LIN {X 0,Y 311.032,Z 352.826,A -85,B 0,C 180,E1 -15949.126,E2 -15949.126} C_VEL
LIN {X 0,Y 312.836,Z 341.868,A -85,B 0,C 180,E1 -15950.55,E2 -15950.55} C_VEL
LIN {X 0,Y 314.374,Z 331.182,A -85,B 0,C 180,E1 -15951.646,E2 -15951.646} C_VEL
LIN {X 0,Y 315.929,Z 318.395,A -85,B 0,C 180,E1 -15952.652,E2 -15952.652} C_VEL
LIN {X 0,Y 317.171,Z 305.489,A -85,B 0,C 180,E1 -15953.377,E2 -15953.377} C_VEL
LIN {X 0,Y 317.99,Z 291.946,A -85,B 0,C 180,E1 -15953.864,E2 -15953.864} C_VEL
LIN {X 0,Y 319.812,Z 229.515,A -85,B 0,C 180,E1 -15955.377,E2 -15955.377} C_VEL
LIN {X 0,Y 316.738,Z 210.082,A -85,B 0,C 180,E1 -15956.219,E2 -15956.219} C_VEL
LIN {X 0,Y 313.412,Z 194.203,A -85,B 0,C 180,E1 -15957.021,E2 -15957.021} C_VEL
LIN {X 0,Y 310.374,Z 186.88,A -85,B 0,C 180,E1 -15957.598,E2 -15957.598} C_VEL
LIN {X 0,Y 308.319,Z 176.835,A -85,B 0,C 180,E1 -15960.855,E2 -15960.855} C_VEL
LIN {X 0,Y 305.949,Z 167.212,A -85,B 0,C 180,E1 -15964.212,E2 -15964.212} C_VEL
LIN {X 0,Y 305.464,Z 165.436,A -85,B 0,C 180,E1 -15964.901,E2 -15964.901} C_VEL
LIN {X 0,Y 305.434,Z 165.44,A -85,B 0,C 180,E1 -15968.525,E2 -15968.525} C_VEL
LIN {X 0,Y 305.435,Z 165.44,A -85,B 0,C 180,E1 -15972.582,E2 -15972.582} C_VEL
LIN {X 0,Y 305.422,Z 165.442,A -85,B 0,C 180,E1 -15976.344,E2 -15976.344} C_VEL
LIN {X 0,Y 305.411,Z 165.436,A -85,B 0,C 180,E1 -15979.885,E2 -15979.885} C_VEL
LIN {X 0,Y 305.464,Z 165.428,A -85,B 0,C 180,E1 -15983.637,E2 -15983.637} C_VEL
LIN {X 0,Y 305.467,Z 165.428,A -85,B 0,C 180,E1 -15986.483,E2 -15986.483} C_VEL
LIN {X 0,Y 305.419,Z 165.437,A -85,B 0,C 180,E1 -15989.586,E2 -15989.586} C_VEL
LIN {X 0,Y 305.442,Z 165.436,A -85,B 0,C 180,E1 -15992.601,E2 -15992.601} C_VEL
LIN {X 0,Y 305.441,Z 165.427,A -85,B 0,C 180,E1 -15995.533,E2 -15995.533} C_VEL
LIN {X 0,Y 305.475,Z 165.42,A -85,B 0,C 180,E1 -15999.812,E2 -15999.812} C_VEL
LIN {X 0,Y 305.494,Z 165.421,A -85,B 0,C 180,E1 -16003.975,E2 -16003.975} C_VEL
LIN {X 0,Y 305.557,Z 165.423,A -85,B 0,C 180,E1 -16006.703,E2 -16006.703} C_VEL
LIN {X 0,Y 305.766,Z 165.394,A -85,B 0,C 180,E1 -16011.249,E2 -16011.249} C_VEL
LIN {X 0,Y 305.798,Z 165.379,A -85,B 0,C 180,E1 -16013.401,E2 -16013.401} C_VEL
LIN {X 0,Y 305.937,Z 165.369,A -85,B 0,C 180,E1 -16018.684,E2 -16018.684} C_VEL
LIN {X 0,Y 305.937,Z 165.369,A -85,B 0,C 180,E1 -16021.316,E2 -16021.316} C_VEL
LIN {X 0,Y 305.788,Z 165.391,A -85,B 0,C 180,E1 -16026.599,E2 -16026.599} C_VEL
LIN {X 0,Y 305.697,Z 165.4,A -85,B 0,C 180,E1 -16029.261,E2 -16029.261} C_VEL
LIN {X 0,Y 305.573,Z 165.418,A -85,B 0,C 180,E1 -16033.297,E2 -16033.297} C_VEL
LIN {X 0,Y 305.514,Z 165.427,A -85,B 0,C 180,E1 -16036.025,E2 -16036.025} C_VEL
LIN {X 0,Y 305.475,Z 165.431,A -85,B 0,C 180,E1 -16040.188,E2 -16040.188} C_VEL
LIN {X 0,Y 305.443,Z 165.439,A -85,B 0,C 180,E1 -16044.467,E2 -16044.467} C_VEL
LIN {X 0,Y 305.454,Z 165.451,A -85,B 0,C 180,E1 -16047.213,E2 -16047.213} C_VEL
LIN {X 0,Y 307.467,Z 173.471,A -85,B 0,C 180,E1 -16050.15,E2 -16050.15} C_VEL
LIN {X 0,Y 315.579,Z 190.715,A -85,B 0,C 180,E1 -16051.565,E2 -16051.565} C_VEL
LIN {X 0,Y 319.554,Z 201.138,A -85,B 0,C 180,E1 -16052.271,E2 -16052.271} C_VEL
LIN {X 0,Y 320.576,Z 206.188,A -85,B 0,C 180,E1 -16052.511,E2 -16052.511} C_VEL
LIN {X 0,Y 318.103,Z 281.171,A -85,B 0,C 180,E1 -16054.335,E2 -16054.335} C_VEL
LIN {X 0,Y 317.204,Z 294.383,A -85,B 0,C 180,E1 -16054.902,E2 -16054.902} C_VEL
LIN {X 0,Y 316.114,Z 307.547,A -85,B 0,C 180,E1 -16055.758,E2 -16055.758} C_VEL
LIN {X 0,Y 314.765,Z 318.834,A -85,B 0,C 180,E1 -16056.743,E2 -16056.743} C_VEL
LIN {X 0,Y 313.128,Z 330.027,A -85,B 0,C 180,E1 -16057.991,E2 -16057.991} C_VEL
LIN {X 0,Y 311.462,Z 340.557,A -85,B 0,C 180,E1 -16059.476,E2 -16059.476} C_VEL
LIN {X 0,Y 309.82,Z 349.922,A -85,B 0,C 180,E1 -16061.136,E2 -16061.136} C_VEL
LIN {X 0,Y 308.123,Z 358.925,A -85,B 0,C 180,E1 -16063.122,E2 -16063.122} C_VEL
LIN {X 0,Y 306.651,Z 366.582,A -85,B 0,C 180,E1 -16065.274,E2 -16065.274} C_VEL
LIN {X 0,Y 305.538,Z 372.451,A -85,B 0,C 180,E1 -16067.398,E2 -16067.398} C_VEL
LIN {X 0,Y 304.642,Z 377.4,A -85,B 0,C 180,E1 -16069.762,E2 -16069.762} C_VEL
LIN {X 0,Y 304.056,Z 380.454,A -85,B 0,C 180,E1 -16071.803,E2 -16071.803} C_VEL
LIN {X 0,Y 303.595,Z 382.701,A -85,B 0,C 180,E1 -16074.118,E2 -16074.118} C_VEL
LIN {X 0,Y 303.326,Z 383.694,A -85,B 0,C 180,E1 -16076.524,E2 -16076.524} C_VEL
LIN {X 0,Y 303.317,Z 383.355,A -85,B 0,C 180,E1 -16079.016,E2 -16079.016} C_VEL
LIN {X 0,Y 303.5,Z 381.483,A -85,B 0,C 180,E1 -16081.637,E2 -16081.637} C_VEL
LIN {X 0,Y 303.941,Z 378.457,A -85,B 0,C 180,E1 -16083.938,E2 -16083.938} C_VEL
LIN {X 0,Y 304.435,Z 374.226,A -85,B 0,C 180,E1 -16086.172,E2 -16086.172} C_VEL
LIN {X 0,Y 305.054,Z 368.671,A -85,B 0,C 180,E1 -16088.369,E2 -16088.369} C_VEL
LIN {X 0,Y 305.932,Z 362.172,A -85,B 0,C 180,E1 -16090.369,E2 -16090.369} C_VEL
LIN {X 0,Y 307.109,Z 354.061,A -85,B 0,C 180,E1 -16092.349,E2 -16092.349} C_VEL
LIN {X 0,Y 308.333,Z 345.04,A -85,B 0,C 180,E1 -16094.126,E2 -16094.126} C_VEL
LIN {X 0,Y 309.623,Z 335.151,A -85,B 0,C 180,E1 -16095.694,E2 -16095.694} C_VEL
LIN {X 0,Y 310.97,Z 323.96,A -85,B 0,C 180,E1 -16097.104,E2 -16097.104} C_VEL
LIN {X 0,Y 312.192,Z 311.78,A -85,B 0,C 180,E1 -16098.31,E2 -16098.31} C_VEL
LIN {X 0,Y 313.171,Z 299.062,A -85,B 0,C 180,E1 -16099.249,E2 -16099.249} C_VEL
LIN {X 0,Y 314.061,Z 285.587,A -85,B 0,C 180,E1 -16099.942,E2 -16099.942} C_VEL
LIN {X 0,Y 314.631,Z 272.038,A -85,B 0,C 180,E1 -16100.359,E2 -16100.359} C_VEL
LIN {X 0,Y 316.256,Z 204.158,A -85,B 0,C 180,E1 -16101.974,E2 -16101.974} C_VEL
LIN {X 0,Y 313.704,Z 190.916,A -85,B 0,C 180,E1 -16102.495,E2 -16102.495} C_VEL
LIN {X 0,Y 307.202,Z 172.569,A -85,B 0,C 180,E1 -16103.473,E2 -16103.473} C_VEL
LIN {X 0,Y 305.652,Z 165.414,A -85,B 0,C 180,E1 -16105.879,E2 -16105.879} C_VEL
LIN {X 0,Y 305.942,Z 165.377,A -85,B 0,C 180,E1 -16108.684,E2 -16108.684} C_VEL
LIN {X 0,Y 305.949,Z 165.372,A -85,B 0,C 180,E1 -16111.316,E2 -16111.316} C_VEL
LIN {X 0,Y 305.788,Z 165.394,A -85,B 0,C 180,E1 -16116.599,E2 -16116.599} C_VEL
LIN {X 0,Y 305.7,Z 165.404,A -85,B 0,C 180,E1 -16119.261,E2 -16119.261} C_VEL
LIN {X 0,Y 305.574,Z 165.419,A -85,B 0,C 180,E1 -16123.297,E2 -16123.297} C_VEL
LIN {X 0,Y 305.534,Z 165.421,A -85,B 0,C 180,E1 -16127.399,E2 -16127.399} C_VEL
LIN {X 0,Y 305.497,Z 165.431,A -85,B 0,C 180,E1 -16130.187,E2 -16130.187} C_VEL
LIN {X 0,Y 305.442,Z 165.433,A -85,B 0,C 180,E1 -16134.467,E2 -16134.467} C_VEL
LIN {X 0,Y 305.453,Z 165.436,A -85,B 0,C 180,E1 -16137.398,E2 -16137.398} C_VEL
LIN {X 0,Y 305.432,Z 165.436,A -85,B 0,C 180,E1 -16140.413,E2 -16140.413} C_VEL
LIN {X 0,Y 305.467,Z 165.429,A -85,B 0,C 180,E1 -16144.078,E2 -16144.078} C_VEL
LIN {X 0,Y 305.456,Z 165.432,A -85,B 0,C 180,E1 -16146.742,E2 -16146.742} C_VEL
LIN {X 0,Y 305.411,Z 165.439,A -85,B 0,C 180,E1 -16150.59,E2 -16150.59} C_VEL
LIN {X 0,Y 305.423,Z 165.435,A -85,B 0,C 180,E1 -16153.656,E2 -16153.656} C_VEL
LIN {X 0,Y 305.422,Z 165.433,A -85,B 0,C 180,E1 -16157.707,E2 -16157.707} C_VEL
LIN {X 0,Y 305.462,Z 165.434,A -85,B 0,C 180,E1 -16161.595,E2 -16161.595} C_VEL
LIN {X 0,Y 305.466,Z 165.434,A -85,B 0,C 180,E1 -16163.44,E2 -16163.44} C_VEL
LIN {X 0,Y 304.789,Z 165.52,A -85,B 0,C 180,E1 -16164.541,E2 -16164.541} C_VEL
LIN {X 0,Y 301.922,Z 165.873,A -85,B 0,C 180,E1 -16166.333,E2 -16166.333} C_VEL
LIN {X 0,Y 299.492,Z 166.177,A -85,B 0,C 180,E1 -16167.786,E2 -16167.786} C_VEL
LIN {X 0,Y 298.447,Z 166.308,A -85,B 0,C 180,E1 -16168.913,E2 -16168.913} C_VEL
LIN {X 0,Y 298.361,Z 166.314,A -85,B 0,C 180,E1 -16169.294,E2 -16169.294} C_VEL
LIN {X 0,Y 298.416,Z 166.31,A -85,B 0,C 180,E1 -16171.899,E2 -16171.899} C_VEL
LIN {X 0,Y 298.442,Z 166.309,A -85,B 0,C 180,E1 -16174.92,E2 -16174.92} C_VEL
LIN {X 0,Y 298.401,Z 166.31,A -85,B 0,C 180,E1 -16177.862,E2 -16177.862} C_VEL
LIN {X 0,Y 298.463,Z 166.309,A -85,B 0,C 180,E1 -16180.752,E2 -16180.752} C_VEL
LIN {X 0,Y 298.513,Z 166.296,A -85,B 0,C 180,E1 -16184.991,E2 -16184.991} C_VEL
LIN {X 0,Y 298.585,Z 166.29,A -85,B 0,C 180,E1 -16189.146,E2 -16189.146} C_VEL
LIN {X 0,Y 298.701,Z 166.276,A -85,B 0,C 180,E1 -16191.884,E2 -16191.884} C_VEL
LIN {X 0,Y 298.631,Z 166.284,A -85,B 0,C 180,E1 -16194.598,E2 -16194.598} C_VEL
LIN {X 0,Y 298.906,Z 166.251,A -85,B 0,C 180,E1 -16198.653,E2 -16198.653} C_VEL
LIN {X 0,Y 298.906,Z 166.248,A -85,B 0,C 180,E1 -16201.347,E2 -16201.347} C_VEL
LIN {X 0,Y 298.739,Z 166.26,A -85,B 0,C 180,E1 -16206.755,E2 -16206.755} C_VEL
LIN {X 0,Y 298.627,Z 166.28,A -85,B 0,C 180,E1 -16209.482,E2 -16209.482} C_VEL
LIN {X 0,Y 298.511,Z 166.301,A -85,B 0,C 180,E1 -16213.617,E2 -16213.617} C_VEL
LIN {X 0,Y 298.438,Z 166.307,A -85,B 0,C 180,E1 -16216.415,E2 -16216.415} C_VEL
LIN {X 0,Y 298.431,Z 166.306,A -85,B 0,C 180,E1 -16219.609,E2 -16219.609} C_VEL
LIN {X 0,Y 298.384,Z 166.317,A -85,B 0,C 180,E1 -16223.604,E2 -16223.604} C_VEL
LIN {X 0,Y 298.403,Z 166.312,A -85,B 0,C 180,E1 -16226.583,E2 -16226.583} C_VEL
LIN {X 0,Y 298.359,Z 166.321,A -85,B 0,C 180,E1 -16229.648,E2 -16229.648} C_VEL
LIN {X 0,Y 298.395,Z 166.314,A -85,B 0,C 180,E1 -16232.8,E2 -16232.8} C_VEL
LIN {X 0,Y 298.429,Z 166.311,A -85,B 0,C 180,E1 -16236.802,E2 -16236.802} C_VEL
LIN {X 0,Y 298.375,Z 166.319,A -85,B 0,C 180,E1 -16239.492,E2 -16239.492} C_VEL
LIN {X 0,Y 298.371,Z 166.321,A -85,B 0,C 180,E1 -16243.097,E2 -16243.097} C_VEL
LIN {X 0,Y 298.371,Z 166.318,A -85,B 0,C 180,E1 -16246.915,E2 -16246.915} C_VEL
LIN {X 0,Y 298.385,Z 166.319,A -85,B 0,C 180,E1 -16251.011,E2 -16251.011} C_VEL
LIN {X 0,Y 298.405,Z 166.314,A -85,B 0,C 180,E1 -16253.928,E2 -16253.928} C_VEL
LIN {X 0,Y 298.443,Z 166.428,A -85,B 0,C 180,E1 -16257.421,E2 -16257.421} C_VEL
LIN {X 0,Y 300.766,Z 177.571,A -85,B 0,C 180,E1 -16260.996,E2 -16260.996} C_VEL
LIN {X 0,Y 302.762,Z 188.224,A -85,B 0,C 180,E1 -16264.231,E2 -16264.231} C_VEL
LIN {X 0,Y 307.587,Z 218.337,A -85,B 0,C 180,E1 -16265.396,E2 -16265.396} C_VEL
LIN {X 0,Y 309.155,Z 230.308,A -85,B 0,C 180,E1 -16265.823,E2 -16265.823} C_VEL
LIN {X 0,Y 307.332,Z 297.128,A -85,B 0,C 180,E1 -16267.478,E2 -16267.478} C_VEL
LIN {X 0,Y 306.545,Z 310.661,A -85,B 0,C 180,E1 -16268.082,E2 -16268.082} C_VEL
LIN {X 0,Y 305.404,Z 323.476,A -85,B 0,C 180,E1 -16268.926,E2 -16268.926} C_VEL
LIN {X 0,Y 303.957,Z 336.015,A -85,B 0,C 180,E1 -16270.059,E2 -16270.059} C_VEL
LIN {X 0,Y 302.567,Z 347.245,A -85,B 0,C 180,E1 -16271.374,E2 -16271.374} C_VEL
LIN {X 0,Y 301.134,Z 358.07,A -85,B 0,C 180,E1 -16272.992,E2 -16272.992} C_VEL
LIN {X 0,Y 299.909,Z 367.318,A -85,B 0,C 180,E1 -16274.714,E2 -16274.714} C_VEL
LIN {X 0,Y 298.846,Z 374.721,A -85,B 0,C 180,E1 -16276.398,E2 -16276.398} C_VEL
LIN {X 0,Y 297.823,Z 381.994,A -85,B 0,C 180,E1 -16278.429,E2 -16278.429} C_VEL
LIN {X 0,Y 297.2,Z 387.782,A -85,B 0,C 180,E1 -16280.472,E2 -16280.472} C_VEL
LIN {X 0,Y 296.786,Z 392.321,A -85,B 0,C 180,E1 -16282.516,E2 -16282.516} C_VEL
LIN {X 0,Y 296.552,Z 395.749,A -85,B 0,C 180,E1 -16284.56,E2 -16284.56} C_VEL
LIN {X 0,Y 296.528,Z 397.446,A -85,B 0,C 180,E1 -16285.923,E2 -16285.923} C_VEL
LIN {X 0,Y 296.533,Z 398.73,A -85,B 0,C 180,E1 -16287.283,E2 -16287.283} C_VEL
LIN {X 0,Y 296.494,Z 399.607,A -85,B 0,C 180,E1 -16288.642,E2 -16288.642} C_VEL
LIN {X 0,Y 296.519,Z 400.044,A -85,B 0,C 180,E1 -16290,E2 -16290} C_VEL
LIN {X 0,Y 296.526,Z 399.706,A -85,B 0,C 180,E1 -16292.717,E2 -16292.717} C_VEL
LIN {X 0,Y 296.492,Z 398.949,A -85,B 0,C 180,E1 -16294.078,E2 -16294.078} C_VEL
LIN {X 0,Y 296.546,Z 397.68,A -85,B 0,C 180,E1 -16295.509,E2 -16295.509} C_VEL
LIN {X 0,Y 296.944,Z 394.106,A -85,B 0,C 180,E1 -16298.164,E2 -16298.164} C_VEL
LIN {X 0,Y 297.475,Z 390.176,A -85,B 0,C 180,E1 -16300.206,E2 -16300.206} C_VEL
LIN {X 0,Y 298.313,Z 385.12,A -85,B 0,C 180,E1 -16302.242,E2 -16302.242} C_VEL
LIN {X 0,Y 299.61,Z 378.797,A -85,B 0,C 180,E1 -16304.259,E2 -16304.259} C_VEL
LIN {X 0,Y 301.12,Z 370.91,A -85,B 0,C 180,E1 -16306.265,E2 -16306.265} C_VEL
LIN {X 0,Y 302.543,Z 362.897,A -85,B 0,C 180,E1 -16307.927,E2 -16307.927} C_VEL
LIN {X 0,Y 304.351,Z 353.147,A -85,B 0,C 180,E1 -16309.562,E2 -16309.562} C_VEL
LIN {X 0,Y 306.231,Z 342.338,A -85,B 0,C 180,E1 -16311.014,E2 -16311.014} C_VEL
LIN {X 0,Y 307.826,Z 331.832,A -85,B 0,C 180,E1 -16312.13,E2 -16312.13} C_VEL
LIN {X 0,Y 309.437,Z 319.276,A -85,B 0,C 180,E1 -16313.154,E2 -16313.154} C_VEL
LIN {X 0,Y 310.789,Z 306.1,A -85,B 0,C 180,E1 -16313.931,E2 -16313.931} C_VEL
LIN {X 0,Y 311.658,Z 292.638,A -85,B 0,C 180,E1 -16314.439,E2 -16314.439} C_VEL
LIN {X 0,Y 313.519,Z 229.757,A -85,B 0,C 180,E1 -16316.005,E2 -16316.005} C_VEL
LIN {X 0,Y 310.646,Z 211.614,A -85,B 0,C 180,E1 -16316.829,E2 -16316.829} C_VEL
LIN {X 0,Y 307.75,Z 197.373,A -85,B 0,C 180,E1 -16317.565,E2 -16317.565} C_VEL
LIN {X 0,Y 303.156,Z 186.693,A -85,B 0,C 180,E1 -16318.437,E2 -16318.437} C_VEL
LIN {X 0,Y 301.15,Z 177.089,A -85,B 0,C 180,E1 -16321.674,E2 -16321.674} C_VEL
LIN {X 0,Y 299.077,Z 168.828,A -85,B 0,C 180,E1 -16324.668,E2 -16324.668} C_VEL
LIN {X 0,Y 298.409,Z 166.316,A -85,B 0,C 180,E1 -16325.664,E2 -16325.664} C_VEL
LIN {X 0,Y 298.375,Z 166.319,A -85,B 0,C 180,E1 -16329.492,E2 -16329.492} C_VEL
LIN {X 0,Y 298.371,Z 166.324,A -85,B 0,C 180,E1 -16333.097,E2 -16333.097} C_VEL
LIN {X 0,Y 298.371,Z 166.316,A -85,B 0,C 180,E1 -16336.915,E2 -16336.915} C_VEL
LIN {X 0,Y 298.386,Z 166.315,A -85,B 0,C 180,E1 -16341.011,E2 -16341.011} C_VEL
LIN {X 0,Y 298.406,Z 166.309,A -85,B 0,C 180,E1 -16343.928,E2 -16343.928} C_VEL
LIN {X 0,Y 298.395,Z 166.307,A -85,B 0,C 180,E1 -16347.2,E2 -16347.2} C_VEL
LIN {X 0,Y 298.366,Z 166.31,A -85,B 0,C 180,E1 -16350.638,E2 -16350.638} C_VEL
LIN {X 0,Y 298.414,Z 166.302,A -85,B 0,C 180,E1 -16354.918,E2 -16354.918} C_VEL
LIN {X 0,Y 298.391,Z 166.315,A -85,B 0,C 180,E1 -16357.861,E2 -16357.861} C_VEL
LIN {X 0,Y 298.452,Z 166.302,A -85,B 0,C 180,E1 -16360.751,E2 -16360.751} C_VEL
LIN {X 0,Y 298.512,Z 166.292,A -85,B 0,C 180,E1 -16364.991,E2 -16364.991} C_VEL
LIN {X 0,Y 298.58,Z 166.279,A -85,B 0,C 180,E1 -16369.146,E2 -16369.146} C_VEL
LIN {X 0,Y 298.723,Z 166.272,A -85,B 0,C 180,E1 -16371.885,E2 -16371.885} C_VEL
LIN {X 0,Y 298.63,Z 166.278,A -85,B 0,C 180,E1 -16374.598,E2 -16374.598} C_VEL
LIN {X 0,Y 298.905,Z 166.244,A -85,B 0,C 180,E1 -16378.653,E2 -16378.653} C_VEL
LIN {X 0,Y 298.905,Z 166.244,A -85,B 0,C 180,E1 -16381.347,E2 -16381.347} C_VEL
LIN {X 0,Y 298.737,Z 166.27,A -85,B 0,C 180,E1 -16386.755,E2 -16386.755} C_VEL
LIN {X 0,Y 298.628,Z 166.28,A -85,B 0,C 180,E1 -16389.482,E2 -16389.482} C_VEL
LIN {X 0,Y 298.525,Z 166.298,A -85,B 0,C 180,E1 -16393.617,E2 -16393.617} C_VEL
LIN {X 0,Y 298.453,Z 166.309,A -85,B 0,C 180,E1 -16396.414,E2 -16396.414} C_VEL
LIN {X 0,Y 298.432,Z 166.312,A -85,B 0,C 180,E1 -16399.61,E2 -16399.61} C_VEL
LIN {X 0,Y 298.385,Z 166.322,A -85,B 0,C 180,E1 -16403.604,E2 -16403.604} C_VEL
LIN {X 0,Y 298.433,Z 166.461,A -85,B 0,C 180,E1 -16406.505,E2 -16406.505} C_VEL
LIN {X 0,Y 300.353,Z 173.807,A -85,B 0,C 180,E1 -16409.287,E2 -16409.287} C_VEL
LIN {X 0,Y 308.639,Z 190.947,A -85,B 0,C 180,E1 -16410.797,E2 -16410.797} C_VEL
LIN {X 0,Y 313.474,Z 202.882,A -85,B 0,C 180,E1 -16411.679,E2 -16411.679} C_VEL
LIN {X 0,Y 314.388,Z 207.675,A -85,B 0,C 180,E1 -16411.914,E2 -16411.914} C_VEL
LIN {X 0,Y 311.787,Z 281.828,A -85,B 0,C 180,E1 -16413.758,E2 -16413.758} C_VEL
LIN {X 0,Y 310.831,Z 295.256,A -85,B 0,C 180,E1 -16414.354,E2 -16414.354} C_VEL
LIN {X 0,Y 309.692,Z 308.101,A -85,B 0,C 180,E1 -16415.217,E2 -16415.217} C_VEL
LIN {X 0,Y 308.05,Z 320.92,A -85,B 0,C 180,E1 -16416.383,E2 -16416.383} C_VEL
LIN {X 0,Y 306.364,Z 331.94,A -85,B 0,C 180,E1 -16417.681,E2 -16417.681} C_VEL
LIN {X 0,Y 304.695,Z 341.755,A -85,B 0,C 180,E1 -16419.141,E2 -16419.141} C_VEL
LIN {X 0,Y 302.768,Z 351.894,A -85,B 0,C 180,E1 -16421.026,E2 -16421.026} C_VEL
LIN {X 0,Y 301.08,Z 360.5,A -85,B 0,C 180,E1 -16423.052,E2 -16423.052} C_VEL
LIN {X 0,Y 299.557,Z 367.868,A -85,B 0,C 180,E1 -16425.264,E2 -16425.264} C_VEL
LIN {X 0,Y 298.653,Z 372.396,A -85,B 0,C 180,E1 -16426.965,E2 -16426.965} C_VEL
LIN {X 0,Y 297.776,Z 376.795,A -85,B 0,C 180,E1 -16429.048,E2 -16429.048} C_VEL
LIN {X 0,Y 297.108,Z 380.31,A -85,B 0,C 180,E1 -16431.316,E2 -16431.316} C_VEL
LIN {X 0,Y 296.558,Z 382.699,A -85,B 0,C 180,E1 -16433.683,E2 -16433.683} C_VEL
LIN {X 0,Y 296.267,Z 383.861,A -85,B 0,C 180,E1 -16436.127,E2 -16436.127} C_VEL
LIN {X 0,Y 296.213,Z 383.664,A -85,B 0,C 180,E1 -16438.666,E2 -16438.666} C_VEL
LIN {X 0,Y 296.374,Z 381.982,A -85,B 0,C 180,E1 -16441.33,E2 -16441.33} C_VEL
LIN {X 0,Y 296.753,Z 379.745,A -85,B 0,C 180,E1 -16443.258,E2 -16443.258} C_VEL
LIN {X 0,Y 297.157,Z 375.953,A -85,B 0,C 180,E1 -16445.55,E2 -16445.55} C_VEL
LIN {X 0,Y 297.793,Z 370.814,A -85,B 0,C 180,E1 -16447.814,E2 -16447.814} C_VEL
LIN {X 0,Y 298.563,Z 364.919,A -85,B 0,C 180,E1 -16449.828,E2 -16449.828} C_VEL
LIN {X 0,Y 299.668,Z 357.311,A -85,B 0,C 180,E1 -16451.896,E2 -16451.896} C_VEL
LIN {X 0,Y 300.898,Z 348.956,A -85,B 0,C 180,E1 -16453.723,E2 -16453.723} C_VEL
LIN {X 0,Y 302.146,Z 339.804,A -85,B 0,C 180,E1 -16455.347,E2 -16455.347} C_VEL
LIN {X 0,Y 303.499,Z 329.746,A -85,B 0,C 180,E1 -16456.785,E2 -16456.785} C_VEL
LIN {X 0,Y 304.724,Z 319.031,A -85,B 0,C 180,E1 -16458.02,E2 -16458.02} C_VEL
LIN {X 0,Y 305.805,Z 307.466,A -85,B 0,C 180,E1 -16459.07,E2 -16459.07} C_VEL
LIN {X 0,Y 306.774,Z 294.987,A -85,B 0,C 180,E1 -16459.911,E2 -16459.911} C_VEL
LIN {X 0,Y 307.587,Z 281.218,A -85,B 0,C 180,E1 -16460.532,E2 -16460.532} C_VEL
LIN {X 0,Y 308.714,Z 240.672,A -85,B 0,C 180,E1 -16461.552,E2 -16461.552} C_VEL
LIN {X 0,Y 309.537,Z 204.633,A -85,B 0,C 180,E1 -16462.437,E2 -16462.437} C_VEL
LIN {X 0,Y 307.225,Z 192.932,A -85,B 0,C 180,E1 -16462.916,E2 -16462.916} C_VEL
LIN {X 0,Y 300.02,Z 172.809,A -85,B 0,C 180,E1 -16464.021,E2 -16464.021} C_VEL
LIN {X 0,Y 298.651,Z 166.289,A -85,B 0,C 180,E1 -16466.289,E2 -16466.289} C_VEL
LIN {X 0,Y 298.911,Z 166.253,A -85,B 0,C 180,E1 -16468.653,E2 -16468.653} C_VEL
LIN {X 0,Y 298.915,Z 166.248,A -85,B 0,C 180,E1 -16471.347,E2 -16471.347} C_VEL
LIN {X 0,Y 298.737,Z 166.272,A -85,B 0,C 180,E1 -16476.755,E2 -16476.755} C_VEL
LIN {X 0,Y 298.633,Z 166.285,A -85,B 0,C 180,E1 -16479.482,E2 -16479.482} C_VEL
LIN {X 0,Y 298.526,Z 166.298,A -85,B 0,C 180,E1 -16483.617,E2 -16483.617} C_VEL
LIN {X 0,Y 298.467,Z 166.302,A -85,B 0,C 180,E1 -16486.413,E2 -16486.413} C_VEL
LIN {X 0,Y 298.48,Z 166.305,A -85,B 0,C 180,E1 -16489.637,E2 -16489.637} C_VEL
LIN {X 0,Y 298.384,Z 166.315,A -85,B 0,C 180,E1 -16493.604,E2 -16493.604} C_VEL
LIN {X 0,Y 298.405,Z 166.311,A -85,B 0,C 180,E1 -16496.583,E2 -16496.583} C_VEL
LIN {X 0,Y 298.395,Z 166.317,A -85,B 0,C 180,E1 -16499.644,E2 -16499.644} C_VEL
LIN {X 0,Y 298.395,Z 166.308,A -85,B 0,C 180,E1 -16502.801,E2 -16502.801} C_VEL
LIN {X 0,Y 298.43,Z 166.307,A -85,B 0,C 180,E1 -16506.803,E2 -16506.803} C_VEL
LIN {X 0,Y 298.376,Z 166.32,A -85,B 0,C 180,E1 -16509.492,E2 -16509.492} C_VEL
LIN {X 0,Y 298.373,Z 166.317,A -85,B 0,C 180,E1 -16513.098,E2 -16513.098} C_VEL
LIN {X 0,Y 298.372,Z 166.307,A -85,B 0,C 180,E1 -16516.915,E2 -16516.915} C_VEL
LIN {X 0,Y 298.387,Z 166.315,A -85,B 0,C 180,E1 -16521.011,E2 -16521.011} C_VEL
LIN {X 0,Y 298.407,Z 166.312,A -85,B 0,C 180,E1 -16523.928,E2 -16523.928} C_VEL
LIN {X 0,Y 298.395,Z 166.313,A -85,B 0,C 180,E1 -16527.2,E2 -16527.2} C_VEL
LIN {X 0,Y 298.361,Z 166.314,A -85,B 0,C 180,E1 -16529.294,E2 -16529.294} C_VEL
LIN {X 0,Y 297.686,Z 166.403,A -85,B 0,C 180,E1 -16530.422,E2 -16530.422} C_VEL
LIN {X 0,Y 294.83,Z 166.758,A -85,B 0,C 180,E1 -16532.258,E2 -16532.258} C_VEL
LIN {X 0,Y 292.425,Z 167.056,A -85,B 0,C 180,E1 -16533.749,E2 -16533.749} C_VEL
LIN {X 0,Y 291.411,Z 167.184,A -85,B 0,C 180,E1 -16534.903,E2 -16534.903} C_VEL
LIN {X 0,Y 291.339,Z 167.187,A -85,B 0,C 180,E1 -16535.294,E2 -16535.294} C_VEL
LIN {X 0,Y 291.348,Z 167.194,A -85,B 0,C 180,E1 -16538.787,E2 -16538.787} C_VEL
LIN {X 0,Y 291.39,Z 167.185,A -85,B 0,C 180,E1 -16541.727,E2 -16541.727} C_VEL
LIN {X 0,Y 291.476,Z 167.175,A -85,B 0,C 180,E1 -16544.683,E2 -16544.683} C_VEL
LIN {X 0,Y 291.531,Z 167.17,A -85,B 0,C 180,E1 -16548.88,E2 -16548.88} C_VEL
LIN {X 0,Y 291.655,Z 167.153,A -85,B 0,C 180,E1 -16551.687,E2 -16551.687} C_VEL
LIN {X 0,Y 291.601,Z 167.16,A -85,B 0,C 180,E1 -16554.468,E2 -16554.468} C_VEL
LIN {X 0,Y 291.874,Z 167.127,A -85,B 0,C 180,E1 -16558.62,E2 -16558.62} C_VEL
LIN {X 0,Y 291.873,Z 167.124,A -85,B 0,C 180,E1 -16561.38,E2 -16561.38} C_VEL
LIN {X 0,Y 291.691,Z 167.136,A -85,B 0,C 180,E1 -16566.919,E2 -16566.919} C_VEL
LIN {X 0,Y 291.569,Z 167.16,A -85,B 0,C 180,E1 -16569.714,E2 -16569.714} C_VEL
LIN {X 0,Y 291.473,Z 167.179,A -85,B 0,C 180,E1 -16573.953,E2 -16573.953} C_VEL
LIN {X 0,Y 291.374,Z 167.183,A -85,B 0,C 180,E1 -16578.274,E2 -16578.274} C_VEL
LIN {X 0,Y 291.341,Z 167.184,A -85,B 0,C 180,E1 -16581.213,E2 -16581.213} C_VEL
LIN {X 0,Y 291.328,Z 167.194,A -85,B 0,C 180,E1 -16584.212,E2 -16584.212} C_VEL
LIN {X 0,Y 291.33,Z 167.196,A -85,B 0,C 180,E1 -16587.281,E2 -16587.281} C_VEL
LIN {X 0,Y 291.304,Z 167.197,A -85,B 0,C 180,E1 -16590.441,E2 -16590.441} C_VEL
LIN {X 0,Y 291.345,Z 167.193,A -85,B 0,C 180,E1 -16593.698,E2 -16593.698} C_VEL
LIN {X 0,Y 291.36,Z 167.194,A -85,B 0,C 180,E1 -16597.249,E2 -16597.249} C_VEL
LIN {X 0,Y 291.301,Z 167.198,A -85,B 0,C 180,E1 -16600.648,E2 -16600.648} C_VEL
LIN {X 0,Y 291.283,Z 167.199,A -85,B 0,C 180,E1 -16604.404,E2 -16604.404} C_VEL
LIN {X 0,Y 291.296,Z 167.199,A -85,B 0,C 180,E1 -16608.411,E2 -16608.411} C_VEL
LIN {X 0,Y 291.335,Z 167.197,A -85,B 0,C 180,E1 -16611.155,E2 -16611.155} C_VEL
LIN {X 0,Y 291.356,Z 167.195,A -85,B 0,C 180,E1 -16614.625,E2 -16614.625} C_VEL
LIN {X 0,Y 291.4,Z 167.287,A -85,B 0,C 180,E1 -16616.991,E2 -16616.991} C_VEL
LIN {X 0,Y 293.718,Z 178.301,A -85,B 0,C 180,E1 -16620.625,E2 -16620.625} C_VEL
LIN {X 0,Y 295.567,Z 188.027,A -85,B 0,C 180,E1 -16623.656,E2 -16623.656} C_VEL
LIN {X 0,Y 296.928,Z 192.982,A -85,B 0,C 180,E1 -16623.902,E2 -16623.902} C_VEL
LIN {X 0,Y 302.282,Z 228.383,A -85,B 0,C 180,E1 -16625.278,E2 -16625.278} C_VEL
LIN {X 0,Y 302.415,Z 235.026,A -85,B 0,C 180,E1 -16625.467,E2 -16625.467} C_VEL
LIN {X 0,Y 300.647,Z 297.039,A -85,B 0,C 180,E1 -16627.04,E2 -16627.04} C_VEL
LIN {X 0,Y 299.808,Z 310.526,A -85,B 0,C 180,E1 -16627.654,E2 -16627.654} C_VEL
LIN {X 0,Y 298.662,Z 323.324,A -85,B 0,C 180,E1 -16628.518,E2 -16628.518} C_VEL
LIN {X 0,Y 297.262,Z 335.061,A -85,B 0,C 180,E1 -16629.59,E2 -16629.59} C_VEL
LIN {X 0,Y 295.781,Z 346.425,A -85,B 0,C 180,E1 -16630.931,E2 -16630.931} C_VEL
LIN {X 0,Y 294.55,Z 355.567,A -85,B 0,C 180,E1 -16632.278,E2 -16632.278} C_VEL
LIN {X 0,Y 293.301,Z 365.087,A -85,B 0,C 180,E1 -16634.004,E2 -16634.004} C_VEL
LIN {X 0,Y 291.932,Z 374.205,A -85,B 0,C 180,E1 -16636.07,E2 -16636.07} C_VEL
LIN {X 0,Y 290.808,Z 381.536,A -85,B 0,C 180,E1 -16638.146,E2 -16638.146} C_VEL
LIN {X 0,Y 290.156,Z 387.393,A -85,B 0,C 180,E1 -16640.238,E2 -16640.238} C_VEL
LIN {X 0,Y 289.715,Z 391.98,A -85,B 0,C 180,E1 -16642.333,E2 -16642.333} C_VEL
LIN {X 0,Y 289.479,Z 395.553,A -85,B 0,C 180,E1 -16644.506,E2 -16644.506} C_VEL
LIN {X 0,Y 289.46,Z 398.47,A -85,B 0,C 180,E1 -16647.217,E2 -16647.217} C_VEL
LIN {X 0,Y 289.415,Z 399.367,A -85,B 0,C 180,E1 -16648.609,E2 -16648.609} C_VEL
LIN {X 0,Y 289.436,Z 399.84,A -85,B 0,C 180,E1 -16650,E2 -16650} C_VEL
LIN {X 0,Y 289.407,Z 399.883,A -85,B 0,C 180,E1 -16651.392,E2 -16651.392} C_VEL
LIN {X 0,Y 289.429,Z 399.535,A -85,B 0,C 180,E1 -16652.784,E2 -16652.784} C_VEL
LIN {X 0,Y 289.428,Z 397.82,A -85,B 0,C 180,E1 -16655.388,E2 -16655.388} C_VEL
LIN {X 0,Y 289.731,Z 395.113,A -85,B 0,C 180,E1 -16657.667,E2 -16657.667} C_VEL
LIN {X 0,Y 290.256,Z 391.583,A -85,B 0,C 180,E1 -16659.758,E2 -16659.758} C_VEL
LIN {X 0,Y 291.046,Z 386.969,A -85,B 0,C 180,E1 -16661.844,E2 -16661.844} C_VEL
LIN {X 0,Y 292.482,Z 380.004,A -85,B 0,C 180,E1 -16664.259,E2 -16664.259} C_VEL
LIN {X 0,Y 294.034,Z 372.485,A -85,B 0,C 180,E1 -16666.311,E2 -16666.311} C_VEL
LIN {X 0,Y 295.466,Z 364.842,A -85,B 0,C 180,E1 -16668.012,E2 -16668.012} C_VEL
LIN {X 0,Y 297.268,Z 355.601,A -85,B 0,C 180,E1 -16669.688,E2 -16669.688} C_VEL
LIN {X 0,Y 299.172,Z 345.347,A -85,B 0,C 180,E1 -16671.173,E2 -16671.173} C_VEL
LIN {X 0,Y 301.073,Z 334.023,A -85,B 0,C 180,E1 -16672.473,E2 -16672.473} C_VEL
LIN {X 0,Y 302.702,Z 322.337,A -85,B 0,C 180,E1 -16673.519,E2 -16673.519} C_VEL
LIN {X 0,Y 304.124,Z 309.655,A -85,B 0,C 180,E1 -16674.353,E2 -16674.353} C_VEL
LIN {X 0,Y 305.277,Z 295.79,A -85,B 0,C 180,E1 -16674.961,E2 -16674.961} C_VEL
LIN {X 0,Y 307.399,Z 230.992,A -85,B 0,C 180,E1 -16676.629,E2 -16676.629} C_VEL
LIN {X 0,Y 304.503,Z 212.687,A -85,B 0,C 180,E1 -16677.491,E2 -16677.491} C_VEL
LIN {X 0,Y 301.958,Z 200.192,A -85,B 0,C 180,E1 -16678.16,E2 -16678.16} C_VEL
LIN {X 0,Y 295.935,Z 186.384,A -85,B 0,C 180,E1 -16679.369,E2 -16679.369} C_VEL
LIN {X 0,Y 294.082,Z 177.668,A -85,B 0,C 180,E1 -16682.432,E2 -16682.432} C_VEL
LIN {X 0,Y 291.837,Z 168.977,A -85,B 0,C 180,E1 -16685.732,E2 -16685.732} C_VEL
LIN {X 0,Y 291.383,Z 167.189,A -85,B 0,C 180,E1 -16686.491,E2 -16686.491} C_VEL
LIN {X 0,Y 291.301,Z 167.203,A -85,B 0,C 180,E1 -16690.648,E2 -16690.648} C_VEL
LIN {X 0,Y 291.283,Z 167.201,A -85,B 0,C 180,E1 -16694.404,E2 -16694.404} C_VEL
LIN {X 0,Y 291.296,Z 167.201,A -85,B 0,C 180,E1 -16698.412,E2 -16698.412} C_VEL
LIN {X 0,Y 291.336,Z 167.194,A -85,B 0,C 180,E1 -16701.156,E2 -16701.156} C_VEL
LIN {X 0,Y 291.357,Z 167.191,A -85,B 0,C 180,E1 -16704.625,E2 -16704.625} C_VEL
LIN {X 0,Y 291.368,Z 167.186,A -85,B 0,C 180,E1 -16707.95,E2 -16707.95} C_VEL
LIN {X 0,Y 291.316,Z 167.187,A -85,B 0,C 180,E1 -16711.151,E2 -16711.151} C_VEL
LIN {X 0,Y 291.343,Z 167.186,A -85,B 0,C 180,E1 -16714.265,E2 -16714.265} C_VEL
LIN {X 0,Y 291.351,Z 167.192,A -85,B 0,C 180,E1 -16717.297,E2 -16717.297} C_VEL
LIN {X 0,Y 291.386,Z 167.177,A -85,B 0,C 180,E1 -16720.265,E2 -16720.265} C_VEL
LIN {X 0,Y 291.454,Z 167.169,A -85,B 0,C 180,E1 -16724.699,E2 -16724.699} C_VEL
LIN {X 0,Y 291.524,Z 167.158,A -85,B 0,C 180,E1 -16728.88,E2 -16728.88} C_VEL
LIN {X 0,Y 291.673,Z 167.151,A -85,B 0,C 180,E1 -16731.687,E2 -16731.687} C_VEL
LIN {X 0,Y 291.601,Z 167.152,A -85,B 0,C 180,E1 -16734.468,E2 -16734.468} C_VEL
LIN {X 0,Y 291.872,Z 167.119,A -85,B 0,C 180,E1 -16738.62,E2 -16738.62} C_VEL
LIN {X 0,Y 291.872,Z 167.12,A -85,B 0,C 180,E1 -16741.38,E2 -16741.38} C_VEL
LIN {X 0,Y 291.689,Z 167.149,A -85,B 0,C 180,E1 -16746.919,E2 -16746.919} C_VEL
LIN {X 0,Y 291.571,Z 167.159,A -85,B 0,C 180,E1 -16749.714,E2 -16749.714} C_VEL
LIN {X 0,Y 291.484,Z 167.178,A -85,B 0,C 180,E1 -16753.952,E2 -16753.952} C_VEL
LIN {X 0,Y 291.404,Z 167.188,A -85,B 0,C 180,E1 -16756.823,E2 -16756.823} C_VEL
LIN {X 0,Y 291.394,Z 167.187,A -85,B 0,C 180,E1 -16759.842,E2 -16759.842} C_VEL
LIN {X 0,Y 291.329,Z 167.198,A -85,B 0,C 180,E1 -16764.212,E2 -16764.212} C_VEL
LIN {X 0,Y 291.43,Z 167.396,A -85,B 0,C 180,E1 -16765.727,E2 -16765.727} C_VEL
LIN {X 0,Y 293.1,Z 173.949,A -85,B 0,C 180,E1 -16768.335,E2 -16768.335} C_VEL
LIN {X 0,Y 300.864,Z 189.498,A -85,B 0,C 180,E1 -16769.832,E2 -16769.832} C_VEL
LIN {X 0,Y 306.543,Z 202.63,A -85,B 0,C 180,E1 -16770.897,E2 -16770.897} C_VEL
LIN {X 0,Y 307.991,Z 207.299,A -85,B 0,C 180,E1 -16771.198,E2 -16771.198} C_VEL
LIN {X 0,Y 308.198,Z 209.901,A -85,B 0,C 180,E1 -16771.297,E2 -16771.297} C_VEL
LIN {X 0,Y 305.555,Z 281.862,A -85,B 0,C 180,E1 -16773.124,E2 -16773.124} C_VEL
LIN {X 0,Y 304.543,Z 295.462,A -85,B 0,C 180,E1 -16773.739,E2 -16773.739} C_VEL
LIN {X 0,Y 303.469,Z 307.463,A -85,B 0,C 180,E1 -16774.554,E2 -16774.554} C_VEL
LIN {X 0,Y 301.99,Z 318.883,A -85,B 0,C 180,E1 -16775.578,E2 -16775.578} C_VEL
LIN {X 0,Y 300.098,Z 330.727,A -85,B 0,C 180,E1 -16776.948,E2 -16776.948} C_VEL
LIN {X 0,Y 298.312,Z 340.868,A -85,B 0,C 180,E1 -16778.435,E2 -16778.435} C_VEL
LIN {X 0,Y 296.516,Z 350.214,A -85,B 0,C 180,E1 -16780.153,E2 -16780.153} C_VEL
LIN {X 0,Y 294.919,Z 357.78,A -85,B 0,C 180,E1 -16781.855,E2 -16781.855} C_VEL
LIN {X 0,Y 293.275,Z 365.554,A -85,B 0,C 180,E1 -16784.034,E2 -16784.034} C_VEL
LIN {X 0,Y 291.923,Z 371.737,A -85,B 0,C 180,E1 -16786.241,E2 -16786.241} C_VEL
LIN {X 0,Y 290.898,Z 376.564,A -85,B 0,C 180,E1 -16788.5,E2 -16788.5} C_VEL
LIN {X 0,Y 290.101,Z 380.369,A -85,B 0,C 180,E1 -16790.958,E2 -16790.958} C_VEL
LIN {X 0,Y 289.559,Z 382.68,A -85,B 0,C 180,E1 -16793.222,E2 -16793.222} C_VEL
LIN {X 0,Y 289.176,Z 384.061,A -85,B 0,C 180,E1 -16796.014,E2 -16796.014} C_VEL
LIN {X 0,Y 289.099,Z 383.97,A -85,B 0,C 180,E1 -16798.305,E2 -16798.305} C_VEL
LIN {X 0,Y 289.246,Z 382.443,A -85,B 0,C 180,E1 -16801.012,E2 -16801.012} C_VEL
LIN {X 0,Y 289.478,Z 380.94,A -85,B 0,C 180,E1 -16802.53,E2 -16802.53} C_VEL
LIN {X 0,Y 289.934,Z 377.513,A -85,B 0,C 180,E1 -16804.9,E2 -16804.9} C_VEL
LIN {X 0,Y 290.503,Z 372.804,A -85,B 0,C 180,E1 -16807.227,E2 -16807.227} C_VEL
LIN {X 0,Y 291.332,Z 366.814,A -85,B 0,C 180,E1 -16809.483,E2 -16809.483} C_VEL
LIN {X 0,Y 292.274,Z 360.329,A -85,B 0,C 180,E1 -16811.421,E2 -16811.421} C_VEL
LIN {X 0,Y 293.499,Z 352.574,A -85,B 0,C 180,E1 -16813.301,E2 -16813.301} C_VEL
LIN {X 0,Y 294.797,Z 343.102,A -85,B 0,C 180,E1 -16815.15,E2 -16815.15} C_VEL
LIN {X 0,Y 296.285,Z 332.666,A -85,B 0,C 180,E1 -16816.781,E2 -16816.781} C_VEL
LIN {X 0,Y 297.557,Z 322.384,A -85,B 0,C 180,E1 -16818.073,E2 -16818.073} C_VEL
LIN {X 0,Y 298.861,Z 310.035,A -85,B 0,C 180,E1 -16819.281,E2 -16819.281} C_VEL
LIN {X 0,Y 299.905,Z 297.104,A -85,B 0,C 180,E1 -16820.227,E2 -16820.227} C_VEL
LIN {X 0,Y 300.795,Z 284.09,A -85,B 0,C 180,E1 -16820.873,E2 -16820.873} C_VEL
LIN {X 0,Y 301.369,Z 266.657,A -85,B 0,C 180,E1 -16821.381,E2 -16821.381} C_VEL
LIN {X 0,Y 302.941,Z 205.605,A -85,B 0,C 180,E1 -16822.899,E2 -16822.899} C_VEL
LIN {X 0,Y 300.898,Z 195.267,A -85,B 0,C 180,E1 -16823.336,E2 -16823.336} C_VEL
LIN {X 0,Y 293.476,Z 174.928,A -85,B 0,C 180,E1 -16824.488,E2 -16824.488} C_VEL
LIN {X 0,Y 292.761,Z 172.829,A -85,B 0,C 180,E1 -16824.662,E2 -16824.662} C_VEL
LIN {X 0,Y 291.672,Z 167.156,A -85,B 0,C 180,E1 -16826.719,E2 -16826.719} C_VEL
LIN {X 0,Y 291.878,Z 167.129,A -85,B 0,C 180,E1 -16828.62,E2 -16828.62} C_VEL
LIN {X 0,Y 291.882,Z 167.125,A -85,B 0,C 180,E1 -16831.38,E2 -16831.38} C_VEL
LIN {X 0,Y 291.689,Z 167.149,A -85,B 0,C 180,E1 -16836.919,E2 -16836.919} C_VEL
LIN {X 0,Y 291.574,Z 167.166,A -85,B 0,C 180,E1 -16839.714,E2 -16839.714} C_VEL
LIN {X 0,Y 291.485,Z 167.178,A -85,B 0,C 180,E1 -16843.952,E2 -16843.952} C_VEL
LIN {X 0,Y 291.419,Z 167.184,A -85,B 0,C 180,E1 -16848.271,E2 -16848.271} C_VEL
LIN {X 0,Y 291.352,Z 167.191,A -85,B 0,C 180,E1 -16851.213,E2 -16851.213} C_VEL
LIN {X 0,Y 291.329,Z 167.191,A -85,B 0,C 180,E1 -16854.212,E2 -16854.212} C_VEL
LIN {X 0,Y 291.352,Z 167.191,A -85,B 0,C 180,E1 -16857.279,E2 -16857.279} C_VEL
LIN {X 0,Y 291.32,Z 167.193,A -85,B 0,C 180,E1 -16860.439,E2 -16860.439} C_VEL
LIN {X 0,Y 291.346,Z 167.187,A -85,B 0,C 180,E1 -16863.699,E2 -16863.699} C_VEL
LIN {X 0,Y 291.361,Z 167.19,A -85,B 0,C 180,E1 -16867.25,E2 -16867.25} C_VEL
LIN {X 0,Y 291.302,Z 167.197,A -85,B 0,C 180,E1 -16870.648,E2 -16870.648} C_VEL
LIN {X 0,Y 291.283,Z 167.193,A -85,B 0,C 180,E1 -16874.404,E2 -16874.404} C_VEL
LIN {X 0,Y 291.297,Z 167.19,A -85,B 0,C 180,E1 -16878.411,E2 -16878.411} C_VEL
LIN {X 0,Y 291.337,Z 167.194,A -85,B 0,C 180,E1 -16881.156,E2 -16881.156} C_VEL
LIN {X 0,Y 291.357,Z 167.191,A -85,B 0,C 180,E1 -16884.625,E2 -16884.625} C_VEL
LIN {X 0,Y 291.368,Z 167.184,A -85,B 0,C 180,E1 -16887.95,E2 -16887.95} C_VEL
LIN {X 0,Y 291.347,Z 167.194,A -85,B 0,C 180,E1 -16891.154,E2 -16891.154} C_VEL
LIN {X 0,Y 291.361,Z 167.19,A -85,B 0,C 180,E1 -16894.267,E2 -16894.267} C_VEL
LIN {X 0,Y 291.339,Z 167.187,A -85,B 0,C 180,E1 -16895.294,E2 -16895.294} C_VEL
LIN {X 0,Y 290.704,Z 167.271,A -85,B 0,C 180,E1 -16896.448,E2 -16896.448} C_VEL
LIN {X 0,Y 287.882,Z 167.626,A -85,B 0,C 180,E1 -16898.326,E2 -16898.326} C_VEL
LIN {X 0,Y 285.463,Z 167.928,A -85,B 0,C 180,E1 -16899.851,E2 -16899.851} C_VEL
LIN {X 0,Y 284.411,Z 168.057,A -85,B 0,C 180,E1 -16901.032,E2 -16901.032} C_VEL
LIN {X 0,Y 284.319,Z 168.066,A -85,B 0,C 180,E1 -16901.433,E2 -16901.433} C_VEL
LIN {X 0,Y 284.421,Z 168.049,A -85,B 0,C 180,E1 -16905.694,E2 -16905.694} C_VEL
LIN {X 0,Y 284.517,Z 168.044,A -85,B 0,C 180,E1 -16910.043,E2 -16910.043} C_VEL
LIN {X 0,Y 284.645,Z 168.024,A -85,B 0,C 180,E1 -16912.909,E2 -16912.909} C_VEL
LIN {X 0,Y 284.841,Z 168.004,A -85,B 0,C 180,E1 -16918.586,E2 -16918.586} C_VEL
LIN {X 0,Y 284.841,Z 168,A -85,B 0,C 180,E1 -16921.414,E2 -16921.414} C_VEL
LIN {X 0,Y 284.647,Z 168.011,A -85,B 0,C 180,E1 -16927.091,E2 -16927.091} C_VEL
LIN {X 0,Y 284.515,Z 168.04,A -85,B 0,C 180,E1 -16929.957,E2 -16929.957} C_VEL
LIN {X 0,Y 284.408,Z 168.057,A -85,B 0,C 180,E1 -16934.307,E2 -16934.307} C_VEL
LIN {X 0,Y 284.34,Z 168.063,A -85,B 0,C 180,E1 -16937.254,E2 -16937.254} C_VEL
LIN {X 0,Y 284.324,Z 168.057,A -85,B 0,C 180,E1 -16940.246,E2 -16940.246} C_VEL
LIN {X 0,Y 284.295,Z 168.072,A -85,B 0,C 180,E1 -16943.84,E2 -16943.84} C_VEL
LIN {X 0,Y 284.287,Z 168.072,A -85,B 0,C 180,E1 -16947.129,E2 -16947.129} C_VEL
LIN {X 0,Y 284.276,Z 168.073,A -85,B 0,C 180,E1 -16950.084,E2 -16950.084} C_VEL
LIN {X 0,Y 284.306,Z 168.07,A -85,B 0,C 180,E1 -16952.945,E2 -16952.945} C_VEL
LIN {X 0,Y 284.322,Z 168.067,A -85,B 0,C 180,E1 -16956.388,E2 -16956.388} C_VEL
LIN {X 0,Y 284.283,Z 168.072,A -85,B 0,C 180,E1 -16959.999,E2 -16959.999} C_VEL
LIN {X 0,Y 284.235,Z 168.077,A -85,B 0,C 180,E1 -16964.188,E2 -16964.188} C_VEL
LIN {X 0,Y 284.241,Z 168.077,A -85,B 0,C 180,E1 -16968.118,E2 -16968.118} C_VEL
LIN {X 0,Y 284.309,Z 168.07,A -85,B 0,C 180,E1 -16972.282,E2 -16972.282} C_VEL
LIN {X 0,Y 284.342,Z 168.068,A -85,B 0,C 180,E1 -16976.425,E2 -16976.425} C_VEL
LIN {X 0,Y 284.371,Z 168.435,A -85,B 0,C 180,E1 -16976.641,E2 -16976.641} C_VEL
LIN {X 0,Y 286.695,Z 179.116,A -85,B 0,C 180,E1 -16980.265,E2 -16980.265} C_VEL
LIN {X 0,Y 288.298,Z 187.681,A -85,B 0,C 180,E1 -16983.041,E2 -16983.041} C_VEL
LIN {X 0,Y 290.5,Z 194.815,A -85,B 0,C 180,E1 -16983.435,E2 -16983.435} C_VEL
LIN {X 0,Y 295.79,Z 230.4,A -85,B 0,C 180,E1 -16984.848,E2 -16984.848} C_VEL
LIN {X 0,Y 294.022,Z 295.741,A -85,B 0,C 180,E1 -16986.538,E2 -16986.538} C_VEL
LIN {X 0,Y 293.234,Z 308.832,A -85,B 0,C 180,E1 -16987.125,E2 -16987.125} C_VEL
LIN {X 0,Y 292.005,Z 322.086,A -85,B 0,C 180,E1 -16988.003,E2 -16988.003} C_VEL
LIN {X 0,Y 290.598,Z 334.078,A -85,B 0,C 180,E1 -16989.101,E2 -16989.101} C_VEL
LIN {X 0,Y 289.009,Z 345.581,A -85,B 0,C 180,E1 -16990.466,E2 -16990.466} C_VEL
LIN {X 0,Y 287.581,Z 355.987,A -85,B 0,C 180,E1 -16992.03,E2 -16992.03} C_VEL
LIN {X 0,Y 286.183,Z 366.143,A -85,B 0,C 180,E1 -16993.962,E2 -16993.962} C_VEL
LIN {X 0,Y 284.768,Z 375.053,A -85,B 0,C 180,E1 -16996.076,E2 -16996.076} C_VEL
LIN {X 0,Y 283.699,Z 382.159,A -85,B 0,C 180,E1 -16998.207,E2 -16998.207} C_VEL
LIN {X 0,Y 282.942,Z 388.649,A -85,B 0,C 180,E1 -17000.709,E2 -17000.709} C_VEL
LIN {X 0,Y 282.554,Z 392.898,A -85,B 0,C 180,E1 -17002.856,E2 -17002.856} C_VEL
LIN {X 0,Y 282.402,Z 395.472,A -85,B 0,C 180,E1 -17004.54,E2 -17004.54} C_VEL
LIN {X 0,Y 282.365,Z 398.21,A -85,B 0,C 180,E1 -17007.147,E2 -17007.147} C_VEL
LIN {X 0,Y 282.339,Z 399.125,A -85,B 0,C 180,E1 -17008.574,E2 -17008.574} C_VEL
LIN {X 0,Y 282.355,Z 399.632,A -85,B 0,C 180,E1 -17010,E2 -17010} C_VEL
LIN {X 0,Y 282.33,Z 399.696,A -85,B 0,C 180,E1 -17011.426,E2 -17011.426} C_VEL
LIN {X 0,Y 282.335,Z 399.367,A -85,B 0,C 180,E1 -17012.854,E2 -17012.854} C_VEL
LIN {X 0,Y 282.337,Z 397.862,A -85,B 0,C 180,E1 -17015.319,E2 -17015.319} C_VEL
LIN {X 0,Y 282.557,Z 395.956,A -85,B 0,C 180,E1 -17017.144,E2 -17017.144} C_VEL
LIN {X 0,Y 283.032,Z 392.814,A -85,B 0,C 180,E1 -17019.288,E2 -17019.288} C_VEL
LIN {X 0,Y 283.777,Z 388.617,A -85,B 0,C 180,E1 -17021.428,E2 -17021.428} C_VEL
LIN {X 0,Y 285.059,Z 382.234,A -85,B 0,C 180,E1 -17023.909,E2 -17023.909} C_VEL
LIN {X 0,Y 286.694,Z 375.306,A -85,B 0,C 180,E1 -17026.009,E2 -17026.009} C_VEL
LIN {X 0,Y 288.379,Z 366.645,A -85,B 0,C 180,E1 -17028.111,E2 -17028.111} C_VEL
LIN {X 0,Y 290.192,Z 357.87,A -85,B 0,C 180,E1 -17029.82,E2 -17029.82} C_VEL
LIN {X 0,Y 292.356,Z 347.068,A -85,B 0,C 180,E1 -17031.506,E2 -17031.506} C_VEL
LIN {X 0,Y 294.284,Z 336.268,A -85,B 0,C 180,E1 -17032.835,E2 -17032.835} C_VEL
LIN {X 0,Y 296.142,Z 324.232,A -85,B 0,C 180,E1 -17033.98,E2 -17033.98} C_VEL
LIN {X 0,Y 297.64,Z 311.776,A -85,B 0,C 180,E1 -17034.873,E2 -17034.873} C_VEL
LIN {X 0,Y 298.856,Z 298.712,A -85,B 0,C 180,E1 -17035.509,E2 -17035.509} C_VEL
LIN {X 0,Y 299.702,Z 280.483,A -85,B 0,C 180,E1 -17036.037,E2 -17036.037} C_VEL
LIN {X 0,Y 301.288,Z 231.856,A -85,B 0,C 180,E1 -17037.294,E2 -17037.294} C_VEL
LIN {X 0,Y 298.116,Z 211.855,A -85,B 0,C 180,E1 -17038.275,E2 -17038.275} C_VEL
LIN {X 0,Y 296.218,Z 202.851,A -85,B 0,C 180,E1 -17038.792,E2 -17038.792} C_VEL
LIN {X 0,Y 290.142,Z 189.45,A -85,B 0,C 180,E1 -17040.021,E2 -17040.021} C_VEL
LIN {X 0,Y 288.755,Z 186.131,A -85,B 0,C 180,E1 -17040.349,E2 -17040.349} C_VEL
LIN {X 0,Y 286.614,Z 176.812,A -85,B 0,C 180,E1 -17043.801,E2 -17043.801} C_VEL
LIN {X 0,Y 284.322,Z 168.07,A -85,B 0,C 180,E1 -17047.352,E2 -17047.352} C_VEL
LIN {X 0,Y 284.283,Z 168.074,A -85,B 0,C 180,E1 -17049.999,E2 -17049.999} C_VEL
LIN {X 0,Y 284.235,Z 168.079,A -85,B 0,C 180,E1 -17054.188,E2 -17054.188} C_VEL
LIN {X 0,Y 284.241,Z 168.079,A -85,B 0,C 180,E1 -17058.119,E2 -17058.119} C_VEL
LIN {X 0,Y 284.31,Z 168.069,A -85,B 0,C 180,E1 -17062.282,E2 -17062.282} C_VEL
LIN {X 0,Y 284.309,Z 168.07,A -85,B 0,C 180,E1 -17065.351,E2 -17065.351} C_VEL
LIN {X 0,Y 284.28,Z 168.074,A -85,B 0,C 180,E1 -17068.724,E2 -17068.724} C_VEL
LIN {X 0,Y 284.262,Z 168.07,A -85,B 0,C 180,E1 -17071.982,E2 -17071.982} C_VEL
LIN {X 0,Y 284.285,Z 168.061,A -85,B 0,C 180,E1 -17075.148,E2 -17075.148} C_VEL
LIN {X 0,Y 284.298,Z 168.067,A -85,B 0,C 180,E1 -17078.235,E2 -17078.235} C_VEL
LIN {X 0,Y 284.314,Z 168.069,A -85,B 0,C 180,E1 -17081.255,E2 -17081.255} C_VEL
LIN {X 0,Y 284.422,Z 168.044,A -85,B 0,C 180,E1 -17084.513,E2 -17084.513} C_VEL
LIN {X 0,Y 284.455,Z 168.039,A -85,B 0,C 180,E1 -17088.6,E2 -17088.6} C_VEL
LIN {X 0,Y 284.627,Z 168.028,A -85,B 0,C 180,E1 -17091.48,E2 -17091.48} C_VEL
LIN {X 0,Y 284.572,Z 168.026,A -85,B 0,C 180,E1 -17094.331,E2 -17094.331} C_VEL
LIN {X 0,Y 284.839,Z 167.994,A -85,B 0,C 180,E1 -17098.586,E2 -17098.586} C_VEL
LIN {X 0,Y 284.839,Z 167.995,A -85,B 0,C 180,E1 -17101.414,E2 -17101.414} C_VEL
LIN {X 0,Y 284.645,Z 168.027,A -85,B 0,C 180,E1 -17107.091,E2 -17107.091} C_VEL
LIN {X 0,Y 284.516,Z 168.039,A -85,B 0,C 180,E1 -17109.957,E2 -17109.957} C_VEL
LIN {X 0,Y 284.437,Z 168.056,A -85,B 0,C 180,E1 -17114.305,E2 -17114.305} C_VEL
LIN {X 0,Y 284.318,Z 168.067,A -85,B 0,C 180,E1 -17118.744,E2 -17118.744} C_VEL
LIN {X 0,Y 284.298,Z 168.073,A -85,B 0,C 180,E1 -17121.766,E2 -17121.766} C_VEL
LIN {X 0,Y 284.356,Z 168.274,A -85,B 0,C 180,E1 -17124.845,E2 -17124.845} C_VEL
LIN {X 0,Y 285.981,Z 174.379,A -85,B 0,C 180,E1 -17127.342,E2 -17127.342} C_VEL
LIN {X 0,Y 293.98,Z 189.716,A -85,B 0,C 180,E1 -17128.954,E2 -17128.954} C_VEL
LIN {X 0,Y 300.171,Z 203.894,A -85,B 0,C 180,E1 -17130.185,E2 -17130.185} C_VEL
LIN {X 0,Y 302.08,Z 209.428,A -85,B 0,C 180,E1 -17130.579,E2 -17130.579} C_VEL
LIN {X 0,Y 299.387,Z 281.933,A -85,B 0,C 180,E1 -17132.463,E2 -17132.463} C_VEL
LIN {X 0,Y 298.352,Z 295.361,A -85,B 0,C 180,E1 -17133.077,E2 -17133.077} C_VEL
LIN {X 0,Y 297.13,Z 308.237,A -85,B 0,C 180,E1 -17133.969,E2 -17133.969} C_VEL
LIN {X 0,Y 295.551,Z 319.755,A -85,B 0,C 180,E1 -17135.036,E2 -17135.036} C_VEL
LIN {X 0,Y 293.664,Z 330.969,A -85,B 0,C 180,E1 -17136.366,E2 -17136.366} C_VEL
LIN {X 0,Y 291.783,Z 341.101,A -85,B 0,C 180,E1 -17137.884,E2 -17137.884} C_VEL
LIN {X 0,Y 289.868,Z 350.55,A -85,B 0,C 180,E1 -17139.664,E2 -17139.664} C_VEL
LIN {X 0,Y 288.111,Z 358.441,A -85,B 0,C 180,E1 -17141.496,E2 -17141.496} C_VEL
LIN {X 0,Y 286.649,Z 364.966,A -85,B 0,C 180,E1 -17143.354,E2 -17143.354} C_VEL
LIN {X 0,Y 285.179,Z 371.328,A -85,B 0,C 180,E1 -17145.617,E2 -17145.617} C_VEL
LIN {X 0,Y 283.985,Z 376.591,A -85,B 0,C 180,E1 -17148.072,E2 -17148.072} C_VEL
LIN {X 0,Y 283.209,Z 380.075,A -85,B 0,C 180,E1 -17150.29,E2 -17150.29} C_VEL
LIN {X 0,Y 282.544,Z 382.679,A -85,B 0,C 180,E1 -17152.747,E2 -17152.747} C_VEL
LIN {X 0,Y 282.138,Z 384.092,A -85,B 0,C 180,E1 -17155.288,E2 -17155.288} C_VEL
LIN {X 0,Y 282.008,Z 384.234,A -85,B 0,C 180,E1 -17157.922,E2 -17157.922} C_VEL
LIN {X 0,Y 282.115,Z 382.895,A -85,B 0,C 180,E1 -17160.682,E2 -17160.682} C_VEL
LIN {X 0,Y 282.586,Z 379.879,A -85,B 0,C 180,E1 -17163.552,E2 -17163.552} C_VEL
LIN {X 0,Y 283.046,Z 376.239,A -85,B 0,C 180,E1 -17165.814,E2 -17165.814} C_VEL
LIN {X 0,Y 283.696,Z 371.065,A -85,B 0,C 180,E1 -17168.186,E2 -17168.186} C_VEL
LIN {X 0,Y 284.712,Z 364.161,A -85,B 0,C 180,E1 -17170.601,E2 -17170.601} C_VEL
LIN {X 0,Y 286.059,Z 355.916,A -85,B 0,C 180,E1 -17172.853,E2 -17172.853} C_VEL
LIN {X 0,Y 287.359,Z 347.146,A -85,B 0,C 180,E1 -17174.757,E2 -17174.757} C_VEL
LIN {X 0,Y 288.672,Z 338.232,A -85,B 0,C 180,E1 -17176.333,E2 -17176.333} C_VEL
LIN {X 0,Y 290.244,Z 326.914,A -85,B 0,C 180,E1 -17177.945,E2 -17177.945} C_VEL
LIN {X 0,Y 291.54,Z 315.53,A -85,B 0,C 180,E1 -17179.211,E2 -17179.211} C_VEL
LIN {X 0,Y 292.775,Z 302.399,A -85,B 0,C 180,E1 -17180.326,E2 -17180.326} C_VEL
LIN {X 0,Y 293.761,Z 289.483,A -85,B 0,C 180,E1 -17181.097,E2 -17181.097} C_VEL
LIN {X 0,Y 294.443,Z 276.474,A -85,B 0,C 180,E1 -17181.593,E2 -17181.593} C_VEL
LIN {X 0,Y 296.409,Z 206.927,A -85,B 0,C 180,E1 -17183.363,E2 -17183.363} C_VEL
LIN {X 0,Y 294.526,Z 197.481,A -85,B 0,C 180,E1 -17183.772,E2 -17183.772} C_VEL
LIN {X 0,Y 287.51,Z 178.107,A -85,B 0,C 180,E1 -17184.898,E2 -17184.898} C_VEL
LIN {X 0,Y 285.59,Z 173.143,A -85,B 0,C 180,E1 -17185.231,E2 -17185.231} C_VEL
LIN {X 0,Y 284.692,Z 168.025,A -85,B 0,C 180,E1 -17187.081,E2 -17187.081} C_VEL
LIN {X 0,Y 284.83,Z 168.007,A -85,B 0,C 180,E1 -17190,E2 -17190} C_VEL
LIN {X 0,Y 284.72,Z 168.017,A -85,B 0,C 180,E1 -17192.83,E2 -17192.83} C_VEL
LIN {X 0,Y 284.645,Z 168.026,A -85,B 0,C 180,E1 -17197.091,E2 -17197.091} C_VEL
LIN {X 0,Y 284.519,Z 168.046,A -85,B 0,C 180,E1 -17199.957,E2 -17199.957} C_VEL
LIN {X 0,Y 284.421,Z 168.056,A -85,B 0,C 180,E1 -17204.306,E2 -17204.306} C_VEL
LIN {X 0,Y 284.361,Z 168.061,A -85,B 0,C 180,E1 -17208.741,E2 -17208.741} C_VEL
LIN {X 0,Y 284.304,Z 168.072,A -85,B 0,C 180,E1 -17211.765,E2 -17211.765} C_VEL
LIN {X 0,Y 284.286,Z 168.066,A -85,B 0,C 180,E1 -17214.852,E2 -17214.852} C_VEL
LIN {X 0,Y 284.283,Z 168.074,A -85,B 0,C 180,E1 -17218.016,E2 -17218.016} C_VEL
LIN {X 0,Y 284.287,Z 168.071,A -85,B 0,C 180,E1 -17221.276,E2 -17221.276} C_VEL
LIN {X 0,Y 284.339,Z 168.06,A -85,B 0,C 180,E1 -17225.347,E2 -17225.347} C_VEL
LIN {X 0,Y 284.3,Z 168.069,A -85,B 0,C 180,E1 -17228.171,E2 -17228.171} C_VEL
LIN {X 0,Y 284.239,Z 168.074,A -85,B 0,C 180,E1 -17232.117,E2 -17232.117} C_VEL
LIN {X 0,Y 284.239,Z 168.062,A -85,B 0,C 180,E1 -17236.186,E2 -17236.186} C_VEL
LIN {X 0,Y 284.285,Z 168.067,A -85,B 0,C 180,E1 -17240.03,E2 -17240.03} C_VEL
LIN {X 0,Y 284.329,Z 168.066,A -85,B 0,C 180,E1 -17243.613,E2 -17243.613} C_VEL
LIN {X 0,Y 284.308,Z 168.067,A -85,B 0,C 180,E1 -17247.19,E2 -17247.19} C_VEL
LIN {X 0,Y 284.339,Z 168.064,A -85,B 0,C 180,E1 -17250.374,E2 -17250.374} C_VEL
LIN {X 0,Y 284.308,Z 168.068,A -85,B 0,C 180,E1 -17253.579,E2 -17253.579} C_VEL
LIN {X 0,Y 284.329,Z 168.065,A -85,B 0,C 180,E1 -17256.704,E2 -17256.704} C_VEL
LIN {X 0,Y 284.325,Z 168.066,A -85,B 0,C 180,E1 -17261.256,E2 -17261.256} C_VEL
LIN {X 0,Y 284.319,Z 168.066,A -85,B 0,C 180,E1 -17261.433,E2 -17261.433} C_VEL
LIN {X 0,Y 283.638,Z 168.155,A -85,B 0,C 180,E1 -17262.616,E2 -17262.616} C_VEL
LIN {X 0,Y 280.81,Z 168.503,A -85,B 0,C 180,E1 -17264.545,E2 -17264.545} C_VEL
LIN {X 0,Y 278.443,Z 168.797,A -85,B 0,C 180,E1 -17266.112,E2 -17266.112} C_VEL
LIN {X 0,Y 277.457,Z 168.92,A -85,B 0,C 180,E1 -17267.325,E2 -17267.325} C_VEL
LIN {X 0,Y 277.392,Z 168.928,A -85,B 0,C 180,E1 -17267.735,E2 -17267.735} C_VEL
LIN {X 0,Y 277.573,Z 168.906,A -85,B 0,C 180,E1 -17271.262,E2 -17271.262} C_VEL
LIN {X 0,Y 277.541,Z 168.91,A -85,B 0,C 180,E1 -17274.186,E2 -17274.186} C_VEL
LIN {X 0,Y 277.808,Z 168.88,A -85,B 0,C 180,E1 -17278.55,E2 -17278.55} C_VEL
LIN {X 0,Y 277.807,Z 168.876,A -85,B 0,C 180,E1 -17281.45,E2 -17281.45} C_VEL
LIN {X 0,Y 277.605,Z 168.887,A -85,B 0,C 180,E1 -17287.272,E2 -17287.272} C_VEL
LIN {X 0,Y 277.454,Z 168.921,A -85,B 0,C 180,E1 -17290.213,E2 -17290.213} C_VEL
LIN {X 0,Y 277.367,Z 168.933,A -85,B 0,C 180,E1 -17294.678,E2 -17294.678} C_VEL
LIN {X 0,Y 277.274,Z 168.938,A -85,B 0,C 180,E1 -17299.239,E2 -17299.239} C_VEL
LIN {X 0,Y 277.257,Z 168.948,A -85,B 0,C 180,E1 -17303.927,E2 -17303.927} C_VEL
LIN {X 0,Y 277.237,Z 168.952,A -85,B 0,C 180,E1 -17307.469,E2 -17307.469} C_VEL
LIN {X 0,Y 277.229,Z 168.95,A -85,B 0,C 180,E1 -17310.465,E2 -17310.465} C_VEL
LIN {X 0,Y 277.247,Z 168.948,A -85,B 0,C 180,E1 -17313.896,E2 -17313.896} C_VEL
LIN {X 0,Y 277.256,Z 168.95,A -85,B 0,C 180,E1 -17317.471,E2 -17317.471} C_VEL
LIN {X 0,Y 277.185,Z 168.958,A -85,B 0,C 180,E1 -17321.241,E2 -17321.241} C_VEL
LIN {X 0,Y 277.175,Z 168.955,A -85,B 0,C 180,E1 -17325.232,E2 -17325.232} C_VEL
LIN {X 0,Y 277.185,Z 168.958,A -85,B 0,C 180,E1 -17328.759,E2 -17328.759} C_VEL
LIN {X 0,Y 277.255,Z 168.949,A -85,B 0,C 180,E1 -17332.528,E2 -17332.528} C_VEL
LIN {X 0,Y 277.306,Z 169.084,A -85,B 0,C 180,E1 -17336.112,E2 -17336.112} C_VEL
LIN {X 0,Y 279.854,Z 180.999,A -85,B 0,C 180,E1 -17340.254,E2 -17340.254} C_VEL
LIN {X 0,Y 281.082,Z 187.659,A -85,B 0,C 180,E1 -17342.425,E2 -17342.425} C_VEL
LIN {X 0,Y 284.085,Z 196.649,A -85,B 0,C 180,E1 -17342.95,E2 -17342.95} C_VEL
LIN {X 0,Y 289.235,Z 231.711,A -85,B 0,C 180,E1 -17344.383,E2 -17344.383} C_VEL
LIN {X 0,Y 287.324,Z 296.418,A -85,B 0,C 180,E1 -17346.101,E2 -17346.101} C_VEL
LIN {X 0,Y 286.432,Z 309.97,A -85,B 0,C 180,E1 -17346.741,E2 -17346.741} C_VEL
LIN {X 0,Y 285.193,Z 322.822,A -85,B 0,C 180,E1 -17347.64,E2 -17347.64} C_VEL
LIN {X 0,Y 283.716,Z 334.584,A -85,B 0,C 180,E1 -17348.76,E2 -17348.76} C_VEL
LIN {X 0,Y 282.097,Z 345.963,A -85,B 0,C 180,E1 -17350.157,E2 -17350.157} C_VEL
LIN {X 0,Y 280.63,Z 356.244,A -85,B 0,C 180,E1 -17351.757,E2 -17351.757} C_VEL
LIN {X 0,Y 279.285,Z 365.653,A -85,B 0,C 180,E1 -17353.591,E2 -17353.591} C_VEL
LIN {X 0,Y 277.866,Z 374.482,A -85,B 0,C 180,E1 -17355.723,E2 -17355.723} C_VEL
LIN {X 0,Y 276.692,Z 381.682,A -85,B 0,C 180,E1 -17357.904,E2 -17357.904} C_VEL
LIN {X 0,Y 275.911,Z 388.232,A -85,B 0,C 180,E1 -17360.47,E2 -17360.47} C_VEL
LIN {X 0,Y 275.492,Z 392.534,A -85,B 0,C 180,E1 -17362.672,E2 -17362.672} C_VEL
LIN {X 0,Y 275.314,Z 395.404,A -85,B 0,C 180,E1 -17364.601,E2 -17364.601} C_VEL
LIN {X 0,Y 275.273,Z 397.939,A -85,B 0,C 180,E1 -17367.073,E2 -17367.073} C_VEL
LIN {X 0,Y 275.264,Z 398.877,A -85,B 0,C 180,E1 -17368.537,E2 -17368.537} C_VEL
LIN {X 0,Y 275.277,Z 399.415,A -85,B 0,C 180,E1 -17370,E2 -17370} C_VEL
LIN {X 0,Y 275.255,Z 399.511,A -85,B 0,C 180,E1 -17371.463,E2 -17371.463} C_VEL
LIN {X 0,Y 275.244,Z 399.202,A -85,B 0,C 180,E1 -17372.927,E2 -17372.927} C_VEL
LIN {X 0,Y 275.3,Z 397.412,A -85,B 0,C 180,E1 -17375.861,E2 -17375.861} C_VEL
LIN {X 0,Y 275.496,Z 395.873,A -85,B 0,C 180,E1 -17377.328,E2 -17377.328} C_VEL
LIN {X 0,Y 275.992,Z 392.774,A -85,B 0,C 180,E1 -17379.528,E2 -17379.528} C_VEL
LIN {X 0,Y 276.789,Z 388.623,A -85,B 0,C 180,E1 -17381.72,E2 -17381.72} C_VEL
LIN {X 0,Y 278.171,Z 382.298,A -85,B 0,C 180,E1 -17384.261,E2 -17384.261} C_VEL
LIN {X 0,Y 279.874,Z 375.443,A -85,B 0,C 180,E1 -17386.41,E2 -17386.41} C_VEL
LIN {X 0,Y 281.554,Z 367.359,A -85,B 0,C 180,E1 -17388.461,E2 -17388.461} C_VEL
LIN {X 0,Y 283.527,Z 358.23,A -85,B 0,C 180,E1 -17390.306,E2 -17390.306} C_VEL
LIN {X 0,Y 285.791,Z 347.537,A -85,B 0,C 180,E1 -17392.026,E2 -17392.026} C_VEL
LIN {X 0,Y 287.783,Z 336.94,A -85,B 0,C 180,E1 -17393.381,E2 -17393.381} C_VEL
LIN {X 0,Y 289.72,Z 325.15,A -85,B 0,C 180,E1 -17394.546,E2 -17394.546} C_VEL
LIN {X 0,Y 291.288,Z 313.025,A -85,B 0,C 180,E1 -17395.453,E2 -17395.453} C_VEL
LIN {X 0,Y 292.614,Z 299.888,A -85,B 0,C 180,E1 -17396.141,E2 -17396.141} C_VEL
LIN {X 0,Y 293.432,Z 284.069,A -85,B 0,C 180,E1 -17396.637,E2 -17396.637} C_VEL
LIN {X 0,Y 295.23,Z 232.79,A -85,B 0,C 180,E1 -17397.989,E2 -17397.989} C_VEL
LIN {X 0,Y 292.337,Z 214.16,A -85,B 0,C 180,E1 -17398.94,E2 -17398.94} C_VEL
LIN {X 0,Y 290.549,Z 205.551,A -85,B 0,C 180,E1 -17399.449,E2 -17399.449} C_VEL
LIN {X 0,Y 284.523,Z 192.349,A -85,B 0,C 180,E1 -17400.718,E2 -17400.718} C_VEL
LIN {X 0,Y 281.549,Z 185.842,A -85,B 0,C 180,E1 -17401.419,E2 -17401.419} C_VEL
LIN {X 0,Y 279.389,Z 176.743,A -85,B 0,C 180,E1 -17404.962,E2 -17404.962} C_VEL
LIN {X 0,Y 277.253,Z 168.95,A -85,B 0,C 180,E1 -17408.316,E2 -17408.316} C_VEL
LIN {X 0,Y 277.193,Z 168.959,A -85,B 0,C 180,E1 -17412.67,E2 -17412.67} C_VEL
LIN {X 0,Y 277.193,Z 168.954,A -85,B 0,C 180,E1 -17416.799,E2 -17416.799} C_VEL
LIN {X 0,Y 277.218,Z 168.948,A -85,B 0,C 180,E1 -17420.669,E2 -17420.669} C_VEL
LIN {X 0,Y 277.28,Z 168.942,A -85,B 0,C 180,E1 -17424.341,E2 -17424.341} C_VEL
LIN {X 0,Y 277.239,Z 168.945,A -85,B 0,C 180,E1 -17427.836,E2 -17427.836} C_VEL
LIN {X 0,Y 277.218,Z 168.943,A -85,B 0,C 180,E1 -17431.204,E2 -17431.204} C_VEL
LIN {X 0,Y 277.233,Z 168.941,A -85,B 0,C 180,E1 -17434.472,E2 -17434.472} C_VEL
LIN {X 0,Y 277.248,Z 168.948,A -85,B 0,C 180,E1 -17437.652,E2 -17437.652} C_VEL
LIN {X 0,Y 277.275,Z 168.939,A -85,B 0,C 180,E1 -17440.761,E2 -17440.761} C_VEL
LIN {X 0,Y 277.367,Z 168.928,A -85,B 0,C 180,E1 -17445.322,E2 -17445.322} C_VEL
LIN {X 0,Y 277.454,Z 168.913,A -85,B 0,C 180,E1 -17449.787,E2 -17449.787} C_VEL
LIN {X 0,Y 277.616,Z 168.892,A -85,B 0,C 180,E1 -17452.728,E2 -17452.728} C_VEL
LIN {X 0,Y 277.806,Z 168.87,A -85,B 0,C 180,E1 -17458.55,E2 -17458.55} C_VEL
LIN {X 0,Y 277.806,Z 168.871,A -85,B 0,C 180,E1 -17461.45,E2 -17461.45} C_VEL
LIN {X 0,Y 277.603,Z 168.905,A -85,B 0,C 180,E1 -17467.272,E2 -17467.272} C_VEL
LIN {X 0,Y 277.456,Z 168.92,A -85,B 0,C 180,E1 -17470.213,E2 -17470.213} C_VEL
LIN {X 0,Y 277.384,Z 168.933,A -85,B 0,C 180,E1 -17474.677,E2 -17474.677} C_VEL
LIN {X 0,Y 277.278,Z 168.947,A -85,B 0,C 180,E1 -17479.239,E2 -17479.239} C_VEL
LIN {X 0,Y 277.289,Z 168.967,A -85,B 0,C 180,E1 -17483.825,E2 -17483.825} C_VEL
LIN {X 0,Y 278.756,Z 174.434,A -85,B 0,C 180,E1 -17486.232,E2 -17486.232} C_VEL
LIN {X 0,Y 287.112,Z 190.174,A -85,B 0,C 180,E1 -17488.032,E2 -17488.032} C_VEL
LIN {X 0,Y 293.826,Z 204.916,A -85,B 0,C 180,E1 -17489.412,E2 -17489.412} C_VEL
LIN {X 0,Y 296.116,Z 210.97,A -85,B 0,C 180,E1 -17489.895,E2 -17489.895} C_VEL
LIN {X 0,Y 293.242,Z 282.128,A -85,B 0,C 180,E1 -17491.778,E2 -17491.778} C_VEL
LIN {X 0,Y 292.131,Z 295.936,A -85,B 0,C 180,E1 -17492.424,E2 -17492.424} C_VEL
LIN {X 0,Y 290.869,Z 308.485,A -85,B 0,C 180,E1 -17493.313,E2 -17493.313} C_VEL
LIN {X 0,Y 289.175,Z 320.288,A -85,B 0,C 180,E1 -17494.431,E2 -17494.431} C_VEL
LIN {X 0,Y 287.125,Z 331.956,A -85,B 0,C 180,E1 -17495.855,E2 -17495.855} C_VEL
LIN {X 0,Y 285.217,Z 341.749,A -85,B 0,C 180,E1 -17497.375,E2 -17497.375} C_VEL
LIN {X 0,Y 283.227,Z 350.951,A -85,B 0,C 180,E1 -17499.155,E2 -17499.155} C_VEL
LIN {X 0,Y 281.528,Z 358.319,A -85,B 0,C 180,E1 -17500.899,E2 -17500.899} C_VEL
LIN {X 0,Y 279.635,Z 366.165,A -85,B 0,C 180,E1 -17503.209,E2 -17503.209} C_VEL
LIN {X 0,Y 278.169,Z 372.201,A -85,B 0,C 180,E1 -17505.483,E2 -17505.483} C_VEL
LIN {X 0,Y 276.929,Z 377.253,A -85,B 0,C 180,E1 -17507.999,E2 -17507.999} C_VEL
LIN {X 0,Y 276.043,Z 380.844,A -85,B 0,C 180,E1 -17510.469,E2 -17510.469} C_VEL
LIN {X 0,Y 275.563,Z 382.684,A -85,B 0,C 180,E1 -17512.258,E2 -17512.258} C_VEL
LIN {X 0,Y 275.084,Z 384.204,A -85,B 0,C 180,E1 -17514.841,E2 -17514.841} C_VEL
LIN {X 0,Y 274.904,Z 384.47,A -85,B 0,C 180,E1 -17517.529,E2 -17517.529} C_VEL
LIN {X 0,Y 275.004,Z 383.338,A -85,B 0,C 180,E1 -17520.332,E2 -17520.332} C_VEL
LIN {X 0,Y 275.431,Z 380.49,A -85,B 0,C 180,E1 -17523.263,E2 -17523.263} C_VEL
LIN {X 0,Y 275.991,Z 376.361,A -85,B 0,C 180,E1 -17525.956,E2 -17525.956} C_VEL
LIN {X 0,Y 276.676,Z 371.156,A -85,B 0,C 180,E1 -17528.388,E2 -17528.388} C_VEL
LIN {X 0,Y 277.705,Z 364.447,A -85,B 0,C 180,E1 -17530.792,E2 -17530.792} C_VEL
LIN {X 0,Y 278.886,Z 357.33,A -85,B 0,C 180,E1 -17532.818,E2 -17532.818} C_VEL
LIN {X 0,Y 280.19,Z 349.077,A -85,B 0,C 180,E1 -17534.73,E2 -17534.73} C_VEL
LIN {X 0,Y 281.747,Z 338.884,A -85,B 0,C 180,E1 -17536.615,E2 -17536.615} C_VEL
LIN {X 0,Y 283.319,Z 328.204,A -85,B 0,C 180,E1 -17538.191,E2 -17538.191} C_VEL
LIN {X 0,Y 284.637,Z 316.997,A -85,B 0,C 180,E1 -17539.508,E2 -17539.508} C_VEL
LIN {X 0,Y 285.909,Z 304.463,A -85,B 0,C 180,E1 -17540.627,E2 -17540.627} C_VEL
LIN {X 0,Y 287.004,Z 291.567,A -85,B 0,C 180,E1 -17541.462,E2 -17541.462} C_VEL
LIN {X 0,Y 287.707,Z 278.479,A -85,B 0,C 180,E1 -17542.014,E2 -17542.014} C_VEL
LIN {X 0,Y 289.751,Z 207.405,A -85,B 0,C 180,E1 -17543.875,E2 -17543.875} C_VEL
LIN {X 0,Y 287.982,Z 199.056,A -85,B 0,C 180,E1 -17544.258,E2 -17544.258} C_VEL
LIN {X 0,Y 280.763,Z 179.38,A -85,B 0,C 180,E1 -17545.453,E2 -17545.453} C_VEL
LIN {X 0,Y 278.394,Z 173.318,A -85,B 0,C 180,E1 -17545.883,E2 -17545.883} C_VEL
LIN {X 0,Y 277.725,Z 168.893,A -85,B 0,C 180,E1 -17547.552,E2 -17547.552} C_VEL
LIN {X 0,Y 277.814,Z 168.877,A -85,B 0,C 180,E1 -17551.45,E2 -17551.45} C_VEL
LIN {X 0,Y 277.603,Z 168.903,A -85,B 0,C 180,E1 -17557.272,E2 -17557.272} C_VEL
LIN {X 0,Y 277.462,Z 168.922,A -85,B 0,C 180,E1 -17560.213,E2 -17560.213} C_VEL
LIN {X 0,Y 277.379,Z 168.931,A -85,B 0,C 180,E1 -17564.677,E2 -17564.677} C_VEL
LIN {X 0,Y 277.317,Z 168.939,A -85,B 0,C 180,E1 -17569.236,E2 -17569.236} C_VEL
LIN {X 0,Y 277.257,Z 168.943,A -85,B 0,C 180,E1 -17573.927,E2 -17573.927} C_VEL
LIN {X 0,Y 277.269,Z 168.947,A -85,B 0,C 180,E1 -17577.482,E2 -17577.482} C_VEL
LIN {X 0,Y 277.25,Z 168.945,A -85,B 0,C 180,E1 -17580.473,E2 -17580.473} C_VEL
LIN {X 0,Y 277.248,Z 168.941,A -85,B 0,C 180,E1 -17583.896,E2 -17583.896} C_VEL
LIN {X 0,Y 277.257,Z 168.949,A -85,B 0,C 180,E1 -17587.471,E2 -17587.471} C_VEL
LIN {X 0,Y 277.186,Z 168.959,A -85,B 0,C 180,E1 -17591.241,E2 -17591.241} C_VEL
LIN {X 0,Y 277.175,Z 168.945,A -85,B 0,C 180,E1 -17595.232,E2 -17595.232} C_VEL
LIN {X 0,Y 277.186,Z 168.947,A -85,B 0,C 180,E1 -17598.759,E2 -17598.759} C_VEL
LIN {X 0,Y 277.262,Z 168.946,A -85,B 0,C 180,E1 -17602.53,E2 -17602.53} C_VEL
LIN {X 0,Y 277.248,Z 168.946,A -85,B 0,C 180,E1 -17606.104,E2 -17606.104} C_VEL
LIN {X 0,Y 277.264,Z 168.945,A -85,B 0,C 180,E1 -17609.539,E2 -17609.539} C_VEL
LIN {X 0,Y 277.295,Z 168.946,A -85,B 0,C 180,E1 -17612.857,E2 -17612.857} C_VEL
LIN {X 0,Y 277.285,Z 168.94,A -85,B 0,C 180,E1 -17616.075,E2 -17616.075} C_VEL
LIN {X 0,Y 277.282,Z 168.947,A -85,B 0,C 180,E1 -17620.762,E2 -17620.762} C_VEL
LIN {X 0,Y 277.374,Z 168.927,A -85,B 0,C 180,E1 -17625.322,E2 -17625.322} C_VEL
LIN {X 0,Y 277.392,Z 168.928,A -85,B 0,C 180,E1 -17627.735,E2 -17627.735} C_VEL
LIN {X 0,Y 276.802,Z 169.007,A -85,B 0,C 180,E1 -17628.948,E2 -17628.948} C_VEL
LIN {X 0,Y 274.094,Z 169.347,A -85,B 0,C 180,E1 -17630.928,E2 -17630.928} C_VEL
LIN {X 0,Y 270.881,Z 169.743,A -85,B 0,C 180,E1 -17633.359,E2 -17633.359} C_VEL
LIN {X 0,Y 270.49,Z 169.786,A -85,B 0,C 180,E1 -17634.199,E2 -17634.199} C_VEL
LIN {X 0,Y 270.773,Z 169.756,A -85,B 0,C 180,E1 -17638.513,E2 -17638.513} C_VEL
LIN {X 0,Y 270.773,Z 169.752,A -85,B 0,C 180,E1 -17641.487,E2 -17641.487} C_VEL
LIN {X 0,Y 270.566,Z 169.763,A -85,B 0,C 180,E1 -17647.462,E2 -17647.462} C_VEL
LIN {X 0,Y 270.386,Z 169.8,A -85,B 0,C 180,E1 -17650.483,E2 -17650.483} C_VEL
LIN {X 0,Y 270.338,Z 169.808,A -85,B 0,C 180,E1 -17655.068,E2 -17655.068} C_VEL
LIN {X 0,Y 270.219,Z 169.812,A -85,B 0,C 180,E1 -17659.762,E2 -17659.762} C_VEL
LIN {X 0,Y 270.184,Z 169.827,A -85,B 0,C 180,E1 -17664.436,E2 -17664.436} C_VEL
LIN {X 0,Y 270.186,Z 169.826,A -85,B 0,C 180,E1 -17667.918,E2 -17667.918} C_VEL
LIN {X 0,Y 270.171,Z 169.834,A -85,B 0,C 180,E1 -17671.35,E2 -17671.35} C_VEL
LIN {X 0,Y 270.2,Z 169.827,A -85,B 0,C 180,E1 -17674.906,E2 -17674.906} C_VEL
LIN {X 0,Y 270.199,Z 169.828,A -85,B 0,C 180,E1 -17678.71,E2 -17678.71} C_VEL
LIN {X 0,Y 270.149,Z 169.835,A -85,B 0,C 180,E1 -17683.245,E2 -17683.245} C_VEL
LIN {X 0,Y 270.152,Z 169.834,A -85,B 0,C 180,E1 -17687.437,E2 -17687.437} C_VEL
LIN {X 0,Y 270.209,Z 169.827,A -85,B 0,C 180,E1 -17691.374,E2 -17691.374} C_VEL
LIN {X 0,Y 270.243,Z 169.84,A -85,B 0,C 180,E1 -17695.591,E2 -17695.591} C_VEL
LIN {X 0,Y 272.782,Z 181.718,A -85,B 0,C 180,E1 -17699.841,E2 -17699.841} C_VEL
LIN {X 0,Y 273.876,Z 187.531,A -85,B 0,C 180,E1 -17701.77,E2 -17701.77} C_VEL
LIN {X 0,Y 277.686,Z 198.344,A -85,B 0,C 180,E1 -17702.442,E2 -17702.442} C_VEL
LIN {X 0,Y 282.647,Z 232.539,A -85,B 0,C 180,E1 -17703.878,E2 -17703.878} C_VEL
LIN {X 0,Y 280.686,Z 295.978,A -85,B 0,C 180,E1 -17705.598,E2 -17705.598} C_VEL
LIN {X 0,Y 279.765,Z 309.603,A -85,B 0,C 180,E1 -17706.251,E2 -17706.251} C_VEL
LIN {X 0,Y 278.467,Z 322.508,A -85,B 0,C 180,E1 -17707.167,E2 -17707.167} C_VEL
LIN {X 0,Y 276.866,Z 335.093,A -85,B 0,C 180,E1 -17708.403,E2 -17708.403} C_VEL
LIN {X 0,Y 275.192,Z 346.345,A -85,B 0,C 180,E1 -17709.832,E2 -17709.832} C_VEL
LIN {X 0,Y 273.865,Z 355.479,A -85,B 0,C 180,E1 -17711.29,E2 -17711.29} C_VEL
LIN {X 0,Y 272.385,Z 365.227,A -85,B 0,C 180,E1 -17713.216,E2 -17713.216} C_VEL
LIN {X 0,Y 270.963,Z 373.911,A -85,B 0,C 180,E1 -17715.351,E2 -17715.351} C_VEL
LIN {X 0,Y 269.718,Z 381.195,A -85,B 0,C 180,E1 -17717.586,E2 -17717.586} C_VEL
LIN {X 0,Y 269.077,Z 386.106,A -85,B 0,C 180,E1 -17719.465,E2 -17719.465} C_VEL
LIN {X 0,Y 268.537,Z 390.858,A -85,B 0,C 180,E1 -17721.724,E2 -17721.724} C_VEL
LIN {X 0,Y 268.249,Z 394.465,A -85,B 0,C 180,E1 -17723.984,E2 -17723.984} C_VEL
LIN {X 0,Y 268.168,Z 396.3,A -85,B 0,C 180,E1 -17725.491,E2 -17725.491} C_VEL
LIN {X 0,Y 268.183,Z 397.667,A -85,B 0,C 180,E1 -17726.996,E2 -17726.996} C_VEL
LIN {X 0,Y 268.191,Z 398.628,A -85,B 0,C 180,E1 -17728.498,E2 -17728.498} C_VEL
LIN {X 0,Y 268.201,Z 399.19,A -85,B 0,C 180,E1 -17730,E2 -17730} C_VEL
LIN {X 0,Y 268.181,Z 399.326,A -85,B 0,C 180,E1 -17731.502,E2 -17731.502} C_VEL
LIN {X 0,Y 268.155,Z 399.037,A -85,B 0,C 180,E1 -17733.005,E2 -17733.005} C_VEL
LIN {X 0,Y 268.225,Z 397.289,A -85,B 0,C 180,E1 -17736.016,E2 -17736.016} C_VEL
LIN {X 0,Y 268.425,Z 395.794,A -85,B 0,C 180,E1 -17737.522,E2 -17737.522} C_VEL
LIN {X 0,Y 268.971,Z 392.746,A -85,B 0,C 180,E1 -17739.779,E2 -17739.779} C_VEL
LIN {X 0,Y 269.819,Z 388.654,A -85,B 0,C 180,E1 -17742.027,E2 -17742.027} C_VEL
LIN {X 0,Y 271.293,Z 382.395,A -85,B 0,C 180,E1 -17744.63,E2 -17744.63} C_VEL
LIN {X 0,Y 273.063,Z 375.602,A -85,B 0,C 180,E1 -17746.831,E2 -17746.831} C_VEL
LIN {X 0,Y 274.706,Z 368.104,A -85,B 0,C 180,E1 -17748.808,E2 -17748.808} C_VEL
LIN {X 0,Y 276.885,Z 358.591,A -85,B 0,C 180,E1 -17750.815,E2 -17750.815} C_VEL
LIN {X 0,Y 279.256,Z 348.005,A -85,B 0,C 180,E1 -17752.569,E2 -17752.569} C_VEL
LIN {X 0,Y 281.314,Z 337.565,A -85,B 0,C 180,E1 -17753.952,E2 -17753.952} C_VEL
LIN {X 0,Y 283.333,Z 326.122,A -85,B 0,C 180,E1 -17755.137,E2 -17755.137} C_VEL
LIN {X 0,Y 285.105,Z 313.126,A -85,B 0,C 180,E1 -17756.144,E2 -17756.144} C_VEL
LIN {X 0,Y 286.486,Z 300.187,A -85,B 0,C 180,E1 -17756.843,E2 -17756.843} C_VEL
LIN {X 0,Y 287.287,Z 286.477,A -85,B 0,C 180,E1 -17757.303,E2 -17757.303} C_VEL
LIN {X 0,Y 289.239,Z 233.97,A -85,B 0,C 180,E1 -17758.713,E2 -17758.713} C_VEL
LIN {X 0,Y 286.404,Z 215.343,A -85,B 0,C 180,E1 -17759.694,E2 -17759.694} C_VEL
LIN {X 0,Y 285.097,Z 208.839,A -85,B 0,C 180,E1 -17760.087,E2 -17760.087} C_VEL
LIN {X 0,Y 278.257,Z 193.686,A -85,B 0,C 180,E1 -17761.618,E2 -17761.618} C_VEL
LIN {X 0,Y 274.332,Z 185.623,A -85,B 0,C 180,E1 -17762.547,E2 -17762.547} C_VEL
LIN {X 0,Y 272.259,Z 177.314,A -85,B 0,C 180,E1 -17765.963,E2 -17765.963} C_VEL
LIN {X 0,Y 270.194,Z 169.83,A -85,B 0,C 180,E1 -17769.347,E2 -17769.347} C_VEL
LIN {X 0,Y 270.149,Z 169.839,A -85,B 0,C 180,E1 -17773.245,E2 -17773.245} C_VEL
LIN {X 0,Y 270.153,Z 169.83,A -85,B 0,C 180,E1 -17777.438,E2 -17777.438} C_VEL
LIN {X 0,Y 270.209,Z 169.828,A -85,B 0,C 180,E1 -17781.374,E2 -17781.374} C_VEL
LIN {X 0,Y 270.2,Z 169.829,A -85,B 0,C 180,E1 -17785.094,E2 -17785.094} C_VEL
LIN {X 0,Y 270.173,Z 169.83,A -85,B 0,C 180,E1 -17789.141,E2 -17789.141} C_VEL
LIN {X 0,Y 270.189,Z 169.824,A -85,B 0,C 180,E1 -17792.177,E2 -17792.177} C_VEL
LIN {X 0,Y 270.184,Z 169.818,A -85,B 0,C 180,E1 -17795.564,E2 -17795.564} C_VEL
LIN {X 0,Y 270.22,Z 169.813,A -85,B 0,C 180,E1 -17800.238,E2 -17800.238} C_VEL
LIN {X 0,Y 270.338,Z 169.8,A -85,B 0,C 180,E1 -17804.932,E2 -17804.932} C_VEL
LIN {X 0,Y 270.386,Z 169.791,A -85,B 0,C 180,E1 -17809.517,E2 -17809.517} C_VEL
LIN {X 0,Y 270.576,Z 169.77,A -85,B 0,C 180,E1 -17812.538,E2 -17812.538} C_VEL
LIN {X 0,Y 270.771,Z 169.745,A -85,B 0,C 180,E1 -17818.513,E2 -17818.513} C_VEL
LIN {X 0,Y 270.771,Z 169.746,A -85,B 0,C 180,E1 -17821.487,E2 -17821.487} C_VEL
LIN {X 0,Y 270.565,Z 169.782,A -85,B 0,C 180,E1 -17827.463,E2 -17827.463} C_VEL
LIN {X 0,Y 270.388,Z 169.803,A -85,B 0,C 180,E1 -17830.483,E2 -17830.483} C_VEL
LIN {X 0,Y 270.347,Z 169.807,A -85,B 0,C 180,E1 -17835.068,E2 -17835.068} C_VEL
LIN {X 0,Y 270.221,Z 169.825,A -85,B 0,C 180,E1 -17839.762,E2 -17839.762} C_VEL
LIN {X 0,Y 270.239,Z 170.002,A -85,B 0,C 180,E1 -17842.86,E2 -17842.86} C_VEL
LIN {X 0,Y 271.607,Z 174.769,A -85,B 0,C 180,E1 -17845.069,E2 -17845.069} C_VEL
LIN {X 0,Y 280.57,Z 191.216,A -85,B 0,C 180,E1 -17847.102,E2 -17847.102} C_VEL
LIN {X 0,Y 286.36,Z 203.553,A -85,B 0,C 180,E1 -17848.366,E2 -17848.366} C_VEL
LIN {X 0,Y 290.161,Z 212.914,A -85,B 0,C 180,E1 -17849.184,E2 -17849.184} C_VEL
LIN {X 0,Y 287.166,Z 282.66,A -85,B 0,C 180,E1 -17851.065,E2 -17851.065} C_VEL
LIN {X 0,Y 286.029,Z 296.049,A -85,B 0,C 180,E1 -17851.704,E2 -17851.704} C_VEL
LIN {X 0,Y 284.707,Z 308.577,A -85,B 0,C 180,E1 -17852.607,E2 -17852.607} C_VEL
LIN {X 0,Y 282.84,Z 320.984,A -85,B 0,C 180,E1 -17853.813,E2 -17853.813} C_VEL
LIN {X 0,Y 280.677,Z 332.608,A -85,B 0,C 180,E1 -17855.273,E2 -17855.273} C_VEL
LIN {X 0,Y 278.565,Z 342.788,A -85,B 0,C 180,E1 -17856.915,E2 -17856.915} C_VEL
LIN {X 0,Y 276.703,Z 351.083,A -85,B 0,C 180,E1 -17858.564,E2 -17858.564} C_VEL
LIN {X 0,Y 274.785,Z 358.88,A -85,B 0,C 180,E1 -17860.456,E2 -17860.456} C_VEL
LIN {X 0,Y 272.813,Z 366.622,A -85,B 0,C 180,E1 -17862.806,E2 -17862.806} C_VEL
LIN {X 0,Y 271.398,Z 372.12,A -85,B 0,C 180,E1 -17864.927,E2 -17864.927} C_VEL
LIN {X 0,Y 270.062,Z 377.119,A -85,B 0,C 180,E1 -17867.42,E2 -17867.42} C_VEL
LIN {X 0,Y 269.032,Z 381.096,A -85,B 0,C 180,E1 -17870.206,E2 -17870.206} C_VEL
LIN {X 0,Y 268.311,Z 383.58,A -85,B 0,C 180,E1 -17872.954,E2 -17872.954} C_VEL
LIN {X 0,Y 268.008,Z 384.435,A -85,B 0,C 180,E1 -17874.766,E2 -17874.766} C_VEL
LIN {X 0,Y 267.805,Z 384.706,A -85,B 0,C 180,E1 -17877.117,E2 -17877.117} C_VEL
LIN {X 0,Y 267.898,Z 383.645,A -85,B 0,C 180,E1 -17880.103,E2 -17880.103} C_VEL
LIN {X 0,Y 268.272,Z 381.096,A -85,B 0,C 180,E1 -17882.963,E2 -17882.963} C_VEL
LIN {X 0,Y 268.731,Z 377.906,A -85,B 0,C 180,E1 -17885.264,E2 -17885.264} C_VEL
LIN {X 0,Y 269.374,Z 373.137,A -85,B 0,C 180,E1 -17887.771,E2 -17887.771} C_VEL
LIN {X 0,Y 270.326,Z 366.955,A -85,B 0,C 180,E1 -17890.246,E2 -17890.246} C_VEL
LIN {X 0,Y 271.561,Z 359.669,A -85,B 0,C 180,E1 -17892.522,E2 -17892.522} C_VEL
LIN {X 0,Y 273.002,Z 350.885,A -85,B 0,C 180,E1 -17894.7,E2 -17894.7} C_VEL
LIN {X 0,Y 274.626,Z 340.877,A -85,B 0,C 180,E1 -17896.684,E2 -17896.684} C_VEL
LIN {X 0,Y 276.14,Z 330.93,A -85,B 0,C 180,E1 -17898.252,E2 -17898.252} C_VEL
LIN {X 0,Y 277.563,Z 320.241,A -85,B 0,C 180,E1 -17899.606,E2 -17899.606} C_VEL
LIN {X 0,Y 278.908,Z 307.877,A -85,B 0,C 180,E1 -17900.833,E2 -17900.833} C_VEL
LIN {X 0,Y 280.018,Z 295.224,A -85,B 0,C 180,E1 -17901.748,E2 -17901.748} C_VEL
LIN {X 0,Y 280.936,Z 281.59,A -85,B 0,C 180,E1 -17902.408,E2 -17902.408} C_VEL
LIN {X 0,Y 283.228,Z 208.733,A -85,B 0,C 180,E1 -17904.377,E2 -17904.377} C_VEL
LIN {X 0,Y 281.775,Z 201.689,A -85,B 0,C 180,E1 -17904.707,E2 -17904.707} C_VEL
LIN {X 0,Y 274.897,Z 182.82,A -85,B 0,C 180,E1 -17905.885,E2 -17905.885} C_VEL
LIN {X 0,Y 271.257,Z 173.551,A -85,B 0,C 180,E1 -17906.528,E2 -17906.528} C_VEL
LIN {X 0,Y 270.713,Z 169.769,A -85,B 0,C 180,E1 -17907.954,E2 -17907.954} C_VEL
LIN {X 0,Y 270.778,Z 169.754,A -85,B 0,C 180,E1 -17911.487,E2 -17911.487} C_VEL
LIN {X 0,Y 270.565,Z 169.78,A -85,B 0,C 180,E1 -17917.462,E2 -17917.462} C_VEL
LIN {X 0,Y 270.413,Z 169.798,A -85,B 0,C 180,E1 -17920.482,E2 -17920.482} C_VEL
LIN {X 0,Y 270.348,Z 169.806,A -85,B 0,C 180,E1 -17925.068,E2 -17925.068} C_VEL
LIN {X 0,Y 270.258,Z 169.822,A -85,B 0,C 180,E1 -17929.759,E2 -17929.759} C_VEL
LIN {X 0,Y 270.179,Z 169.822,A -85,B 0,C 180,E1 -17934.595,E2 -17934.595} C_VEL
LIN {X 0,Y 270.199,Z 169.829,A -85,B 0,C 180,E1 -17937.917,E2 -17937.917} C_VEL
LIN {X 0,Y 270.175,Z 169.828,A -85,B 0,C 180,E1 -17941.35,E2 -17941.35} C_VEL
LIN {X 0,Y 270.2,Z 169.817,A -85,B 0,C 180,E1 -17944.906,E2 -17944.906} C_VEL
LIN {X 0,Y 270.2,Z 169.826,A -85,B 0,C 180,E1 -17948.71,E2 -17948.71} C_VEL
LIN {X 0,Y 270.15,Z 169.828,A -85,B 0,C 180,E1 -17953.245,E2 -17953.245} C_VEL
LIN {X 0,Y 270.153,Z 169.819,A -85,B 0,C 180,E1 -17957.438,E2 -17957.438} C_VEL
LIN {X 0,Y 270.209,Z 169.826,A -85,B 0,C 180,E1 -17961.374,E2 -17961.374} C_VEL
LIN {X 0,Y 270.201,Z 169.828,A -85,B 0,C 180,E1 -17965.094,E2 -17965.094} C_VEL
LIN {X 0,Y 270.186,Z 169.828,A -85,B 0,C 180,E1 -17969.137,E2 -17969.137} C_VEL
LIN {X 0,Y 270.225,Z 169.823,A -85,B 0,C 180,E1 -17972.163,E2 -17972.163} C_VEL
LIN {X 0,Y 270.23,Z 169.818,A -85,B 0,C 180,E1 -17975.543,E2 -17975.543} C_VEL
LIN {X 0,Y 270.224,Z 169.823,A -85,B 0,C 180,E1 -17980.238,E2 -17980.238} C_VEL
LIN {X 0,Y 270.341,Z 169.804,A -85,B 0,C 180,E1 -17984.932,E2 -17984.932} C_VEL
LIN {X 0,Y 270.412,Z 169.799,A -85,B 0,C 180,E1 -17989.518,E2 -17989.518} C_VEL
LIN {X 0,Y 270.565,Z 169.779,A -85,B 0,C 180,E1 -17992.537,E2 -17992.537} C_VEL
LIN {X 0,Y 270.49,Z 169.786,A -85,B 0,C 180,E1 -17994.199,E2 -17994.199} C_VEL
LIN {X 0,Y 269.745,Z 169.88,A -85,B 0,C 180,E1 -17995.444,E2 -17995.444} C_VEL
LIN {X 0,Y 266.991,Z 170.225,A -85,B 0,C 180,E1 -17997.48,E2 -17997.48} C_VEL
LIN {X 0,Y 264.73,Z 170.507,A -85,B 0,C 180,E1 -17999.133,E2 -17999.133} C_VEL
LIN {X 0,Y 263.781,Z 170.625,A -85,B 0,C 180,E1 -18000.411,E2 -18000.411} C_VEL
LIN {X 0,Y 263.71,Z 170.631,A -85,B 0,C 180,E1 -18000.843,E2 -18000.843} C_VEL
LIN {X 0,Y 263.484,Z 170.643,A -85,B 0,C 180,E1 -18006.125,E2 -18006.125} C_VEL
LIN {X 0,Y 263.476,Z 170.653,A -85,B 0,C 180,E1 -18009.266,E2 -18009.266} C_VEL
LIN {X 0,Y 263.251,Z 170.695,A -85,B 0,C 180,E1 -18013.903,E2 -18013.903} C_VEL
LIN {X 0,Y 263.202,Z 170.695,A -85,B 0,C 180,E1 -18017.081,E2 -18017.081} C_VEL
LIN {X 0,Y 263.175,Z 170.687,A -85,B 0,C 180,E1 -18020.825,E2 -18020.825} C_VEL
LIN {X 0,Y 263.122,Z 170.709,A -85,B 0,C 180,E1 -18025.3,E2 -18025.3} C_VEL
LIN {X 0,Y 263.119,Z 170.705,A -85,B 0,C 180,E1 -18028.737,E2 -18028.737} C_VEL
LIN {X 0,Y 263.128,Z 170.707,A -85,B 0,C 180,E1 -18032.289,E2 -18032.289} C_VEL
LIN {X 0,Y 263.177,Z 170.703,A -85,B 0,C 180,E1 -18036.761,E2 -18036.761} C_VEL
LIN {X 0,Y 263.093,Z 170.712,A -85,B 0,C 180,E1 -18039.875,E2 -18039.875} C_VEL
LIN {X 0,Y 263.077,Z 170.712,A -85,B 0,C 180,E1 -18043.994,E2 -18043.994} C_VEL
LIN {X 0,Y 263.082,Z 170.714,A -85,B 0,C 180,E1 -18048.417,E2 -18048.417} C_VEL
LIN {X 0,Y 263.158,Z 170.705,A -85,B 0,C 180,E1 -18052.102,E2 -18052.102} C_VEL
LIN {X 0,Y 263.2,Z 170.726,A -85,B 0,C 180,E1 -18055.093,E2 -18055.093} C_VEL
LIN {X 0,Y 265.71,Z 182.37,A -85,B 0,C 180,E1 -18059.392,E2 -18059.392} C_VEL
LIN {X 0,Y 266.601,Z 187.17,A -85,B 0,C 180,E1 -18061.072,E2 -18061.072} C_VEL
LIN {X 0,Y 271.313,Z 200.329,A -85,B 0,C 180,E1 -18061.927,E2 -18061.927} C_VEL
LIN {X 0,Y 276.063,Z 232.903,A -85,B 0,C 180,E1 -18063.335,E2 -18063.335} C_VEL
LIN {X 0,Y 274.063,Z 295.477,A -85,B 0,C 180,E1 -18065.069,E2 -18065.069} C_VEL
LIN {X 0,Y 273.116,Z 309.193,A -85,B 0,C 180,E1 -18065.737,E2 -18065.737} C_VEL
LIN {X 0,Y 271.789,Z 322.17,A -85,B 0,C 180,E1 -18066.674,E2 -18066.674} C_VEL
LIN {X 0,Y 270.245,Z 333.992,A -85,B 0,C 180,E1 -18067.846,E2 -18067.846} C_VEL
LIN {X 0,Y 268.53,Z 345.413,A -85,B 0,C 180,E1 -18069.309,E2 -18069.309} C_VEL
LIN {X 0,Y 266.932,Z 355.735,A -85,B 0,C 180,E1 -18070.985,E2 -18070.985} C_VEL
LIN {X 0,Y 265.33,Z 365.833,A -85,B 0,C 180,E1 -18073.06,E2 -18073.06} C_VEL
LIN {X 0,Y 263.806,Z 374.704,A -85,B 0,C 180,E1 -18075.34,E2 -18075.34} C_VEL
LIN {X 0,Y 262.562,Z 381.754,A -85,B 0,C 180,E1 -18077.635,E2 -18077.635} C_VEL
LIN {X 0,Y 261.834,Z 387.395,A -85,B 0,C 180,E1 -18079.952,E2 -18079.952} C_VEL
LIN {X 0,Y 261.348,Z 391.802,A -85,B 0,C 180,E1 -18082.273,E2 -18082.273} C_VEL
LIN {X 0,Y 261.124,Z 395.309,A -85,B 0,C 180,E1 -18084.77,E2 -18084.77} C_VEL
LIN {X 0,Y 261.097,Z 397.395,A -85,B 0,C 180,E1 -18086.914,E2 -18086.914} C_VEL
LIN {X 0,Y 261.118,Z 398.378,A -85,B 0,C 180,E1 -18088.458,E2 -18088.458} C_VEL
LIN {X 0,Y 261.127,Z 398.961,A -85,B 0,C 180,E1 -18090,E2 -18090} C_VEL
LIN {X 0,Y 261.108,Z 399.138,A -85,B 0,C 180,E1 -18091.542,E2 -18091.542} C_VEL
LIN {X 0,Y 261.05,Z 398.874,A -85,B 0,C 180,E1 -18093.087,E2 -18093.087} C_VEL
LIN {X 0,Y 261.085,Z 397.943,A -85,B 0,C 180,E1 -18095.137,E2 -18095.137} C_VEL
LIN {X 0,Y 261.361,Z 395.726,A -85,B 0,C 180,E1 -18097.727,E2 -18097.727} C_VEL
LIN {X 0,Y 261.968,Z 392.719,A -85,B 0,C 180,E1 -18100.043,E2 -18100.043} C_VEL
LIN {X 0,Y 262.839,Z 388.677,A -85,B 0,C 180,E1 -18102.352,E2 -18102.352} C_VEL
LIN {X 0,Y 264.427,Z 382.491,A -85,B 0,C 180,E1 -18105.019,E2 -18105.019} C_VEL
LIN {X 0,Y 266.264,Z 375.761,A -85,B 0,C 180,E1 -18107.274,E2 -18107.274} C_VEL
LIN {X 0,Y 268.222,Z 367.416,A -85,B 0,C 180,E1 -18109.53,E2 -18109.53} C_VEL
LIN {X 0,Y 270.275,Z 358.993,A -85,B 0,C 180,E1 -18111.349,E2 -18111.349} C_VEL
LIN {X 0,Y 272.753,Z 348.563,A -85,B 0,C 180,E1 -18113.138,E2 -18113.138} C_VEL
LIN {X 0,Y 275.186,Z 336.885,A -85,B 0,C 180,E1 -18114.721,E2 -18114.721} C_VEL
LIN {X 0,Y 277.25,Z 325.268,A -85,B 0,C 180,E1 -18115.93,E2 -18115.93} C_VEL
LIN {X 0,Y 279.099,Z 312.08,A -85,B 0,C 180,E1 -18116.953,E2 -18116.953} C_VEL
LIN {X 0,Y 280.505,Z 299.672,A -85,B 0,C 180,E1 -18117.614,E2 -18117.614} C_VEL
LIN {X 0,Y 281.384,Z 284.135,A -85,B 0,C 180,E1 -18118.128,E2 -18118.128} C_VEL
LIN {X 0,Y 283.302,Z 235.002,A -85,B 0,C 180,E1 -18119.474,E2 -18119.474} C_VEL
LIN {X 0,Y 280.812,Z 218.08,A -85,B 0,C 180,E1 -18120.394,E2 -18120.394} C_VEL
LIN {X 0,Y 279.53,Z 211.699,A -85,B 0,C 180,E1 -18120.803,E2 -18120.803} C_VEL
LIN {X 0,Y 273.396,Z 197.908,A -85,B 0,C 180,E1 -18122.239,E2 -18122.239} C_VEL
LIN {X 0,Y 268.754,Z 188.857,A -85,B 0,C 180,E1 -18123.353,E2 -18123.353} C_VEL
LIN {X 0,Y 267.05,Z 185.292,A -85,B 0,C 180,E1 -18123.828,E2 -18123.828} C_VEL
LIN {X 0,Y 264.859,Z 176.616,A -85,B 0,C 180,E1 -18127.612,E2 -18127.612} C_VEL
LIN {X 0,Y 263.106,Z 170.714,A -85,B 0,C 180,E1 -18130.499,E2 -18130.499} C_VEL
LIN {X 0,Y 263.078,Z 170.715,A -85,B 0,C 180,E1 -18133.994,E2 -18133.994} C_VEL
LIN {X 0,Y 263.11,Z 170.712,A -85,B 0,C 180,E1 -18138.411,E2 -18138.411} C_VEL
LIN {X 0,Y 263.159,Z 170.705,A -85,B 0,C 180,E1 -18142.103,E2 -18142.103} C_VEL
LIN {X 0,Y 263.153,Z 170.702,A -85,B 0,C 180,E1 -18145.886,E2 -18145.886} C_VEL
LIN {X 0,Y 263.111,Z 170.708,A -85,B 0,C 180,E1 -18149.502,E2 -18149.502} C_VEL
LIN {X 0,Y 263.115,Z 170.71,A -85,B 0,C 180,E1 -18152.994,E2 -18152.994} C_VEL
LIN {X 0,Y 263.117,Z 170.703,A -85,B 0,C 180,E1 -18156.381,E2 -18156.381} C_VEL
LIN {X 0,Y 263.209,Z 170.684,A -85,B 0,C 180,E1 -18159.689,E2 -18159.689} C_VEL
LIN {X 0,Y 263.291,Z 170.675,A -85,B 0,C 180,E1 -18164.518,E2 -18164.518} C_VEL
LIN {X 0,Y 263.33,Z 170.669,A -85,B 0,C 180,E1 -18169.233,E2 -18169.233} C_VEL
LIN {X 0,Y 263.54,Z 170.647,A -85,B 0,C 180,E1 -18172.338,E2 -18172.338} C_VEL
LIN {X 0,Y 263.735,Z 170.621,A -85,B 0,C 180,E1 -18178.473,E2 -18178.473} C_VEL
LIN {X 0,Y 263.735,Z 170.622,A -85,B 0,C 180,E1 -18181.527,E2 -18181.527} C_VEL
LIN {X 0,Y 263.529,Z 170.66,A -85,B 0,C 180,E1 -18187.663,E2 -18187.663} C_VEL
LIN {X 0,Y 263.333,Z 170.684,A -85,B 0,C 180,E1 -18190.767,E2 -18190.767} C_VEL
LIN {X 0,Y 263.293,Z 170.684,A -85,B 0,C 180,E1 -18195.482,E2 -18195.482} C_VEL
LIN {X 0,Y 263.207,Z 170.696,A -85,B 0,C 180,E1 -18200.311,E2 -18200.311} C_VEL
LIN {X 0,Y 263.181,Z 170.811,A -85,B 0,C 180,E1 -18201.708,E2 -18201.708} C_VEL
LIN {X 0,Y 264.465,Z 175.182,A -85,B 0,C 180,E1 -18203.804,E2 -18203.804} C_VEL
LIN {X 0,Y 266.711,Z 179.056,A -85,B 0,C 180,E1 -18204.365,E2 -18204.365} C_VEL
LIN {X 0,Y 273.936,Z 191.972,A -85,B 0,C 180,E1 -18206.088,E2 -18206.088} C_VEL
LIN {X 0,Y 280.122,Z 204.879,A -85,B 0,C 180,E1 -18207.503,E2 -18207.503} C_VEL
LIN {X 0,Y 284.179,Z 214.831,A -85,B 0,C 180,E1 -18208.434,E2 -18208.434} C_VEL
LIN {X 0,Y 281.19,Z 282.498,A -85,B 0,C 180,E1 -18210.293,E2 -18210.293} C_VEL
LIN {X 0,Y 279.96,Z 296.447,A -85,B 0,C 180,E1 -18210.968,E2 -18210.968} C_VEL
LIN {X 0,Y 278.604,Z 308.703,A -85,B 0,C 180,E1 -18211.869,E2 -18211.869} C_VEL
LIN {X 0,Y 276.696,Z 320.75,A -85,B 0,C 180,E1 -18213.05,E2 -18213.05} C_VEL
LIN {X 0,Y 274.465,Z 332.406,A -85,B 0,C 180,E1 -18214.531,E2 -18214.531} C_VEL
LIN {X 0,Y 272.256,Z 342.508,A -85,B 0,C 180,E1 -18216.171,E2 -18216.171} C_VEL
LIN {X 0,Y 270.054,Z 351.819,A -85,B 0,C 180,E1 -18218.071,E2 -18218.071} C_VEL
LIN {X 0,Y 268.112,Z 359.268,A -85,B 0,C 180,E1 -18219.938,E2 -18219.938} C_VEL
LIN {X 0,Y 266.073,Z 366.847,A -85,B 0,C 180,E1 -18222.303,E2 -18222.303} C_VEL
LIN {X 0,Y 264.425,Z 372.809,A -85,B 0,C 180,E1 -18224.686,E2 -18224.686} C_VEL
LIN {X 0,Y 263.131,Z 377.4,A -85,B 0,C 180,E1 -18227.071,E2 -18227.071} C_VEL
LIN {X 0,Y 262.017,Z 381.353,A -85,B 0,C 180,E1 -18229.928,E2 -18229.928} C_VEL
LIN {X 0,Y 261.488,Z 383.151,A -85,B 0,C 180,E1 -18231.817,E2 -18231.817} C_VEL
LIN {X 0,Y 261.039,Z 384.394,A -85,B 0,C 180,E1 -18233.872,E2 -18233.872} C_VEL
LIN {X 0,Y 260.765,Z 384.942,A -85,B 0,C 180,E1 -18236.668,E2 -18236.668} C_VEL
LIN {X 0,Y 260.741,Z 384.083,A -85,B 0,C 180,E1 -18239.602,E2 -18239.602} C_VEL
LIN {X 0,Y 261.108,Z 381.675,A -85,B 0,C 180,E1 -18242.652,E2 -18242.652} C_VEL
LIN {X 0,Y 261.64,Z 378.211,A -85,B 0,C 180,E1 -18245.281,E2 -18245.281} C_VEL
LIN {X 0,Y 262.327,Z 373.231,A -85,B 0,C 180,E1 -18247.971,E2 -18247.971} C_VEL
LIN {X 0,Y 263.337,Z 367.017,A -85,B 0,C 180,E1 -18250.512,E2 -18250.512} C_VEL
LIN {X 0,Y 264.663,Z 359.37,A -85,B 0,C 180,E1 -18252.934,E2 -18252.934} C_VEL
LIN {X 0,Y 266.132,Z 350.86,A -85,B 0,C 180,E1 -18255.079,E2 -18255.079} C_VEL
LIN {X 0,Y 267.627,Z 341.781,A -85,B 0,C 180,E1 -18256.932,E2 -18256.932} C_VEL
LIN {X 0,Y 269.4,Z 330.768,A -85,B 0,C 180,E1 -18258.717,E2 -18258.717} C_VEL
LIN {X 0,Y 270.984,Z 318.795,A -85,B 0,C 180,E1 -18260.244,E2 -18260.244} C_VEL
LIN {X 0,Y 272.27,Z 307.352,A -85,B 0,C 180,E1 -18261.371,E2 -18261.371} C_VEL
LIN {X 0,Y 273.414,Z 294.62,A -85,B 0,C 180,E1 -18262.291,E2 -18262.291} C_VEL
LIN {X 0,Y 274.352,Z 281.07,A -85,B 0,C 180,E1 -18262.946,E2 -18262.946} C_VEL
LIN {X 0,Y 276.688,Z 209.74,A -85,B 0,C 180,E1 -18264.911,E2 -18264.911} C_VEL
LIN {X 0,Y 275.456,Z 203.959,A -85,B 0,C 180,E1 -18265.193,E2 -18265.193} C_VEL
LIN {X 0,Y 268.759,Z 185.57,A -85,B 0,C 180,E1 -18266.374,E2 -18266.374} C_VEL
LIN {X 0,Y 264.179,Z 173.699,A -85,B 0,C 180,E1 -18267.236,E2 -18267.236} C_VEL
LIN {X 0,Y 263.746,Z 170.633,A -85,B 0,C 180,E1 -18268.473,E2 -18268.473} C_VEL
LIN {X 0,Y 263.741,Z 170.631,A -85,B 0,C 180,E1 -18271.527,E2 -18271.527} C_VEL
LIN {X 0,Y 263.528,Z 170.658,A -85,B 0,C 180,E1 -18277.663,E2 -18277.663} C_VEL
LIN {X 0,Y 263.352,Z 170.676,A -85,B 0,C 180,E1 -18280.767,E2 -18280.767} C_VEL
LIN {X 0,Y 263.298,Z 170.686,A -85,B 0,C 180,E1 -18285.481,E2 -18285.481} C_VEL
LIN {X 0,Y 263.238,Z 170.695,A -85,B 0,C 180,E1 -18290.309,E2 -18290.309} C_VEL
LIN {X 0,Y 263.128,Z 170.701,A -85,B 0,C 180,E1 -18295.3,E2 -18295.3} C_VEL
LIN {X 0,Y 263.135,Z 170.706,A -85,B 0,C 180,E1 -18298.735,E2 -18298.735} C_VEL
LIN {X 0,Y 263.13,Z 170.698,A -85,B 0,C 180,E1 -18302.289,E2 -18302.289} C_VEL
LIN {X 0,Y 263.178,Z 170.697,A -85,B 0,C 180,E1 -18306.761,E2 -18306.761} C_VEL
LIN {X 0,Y 263.093,Z 170.712,A -85,B 0,C 180,E1 -18309.875,E2 -18309.875} C_VEL
LIN {X 0,Y 263.078,Z 170.703,A -85,B 0,C 180,E1 -18313.994,E2 -18313.994} C_VEL
LIN {X 0,Y 263.082,Z 170.7,A -85,B 0,C 180,E1 -18318.418,E2 -18318.418} C_VEL
LIN {X 0,Y 263.16,Z 170.701,A -85,B 0,C 180,E1 -18322.103,E2 -18322.103} C_VEL
LIN {X 0,Y 263.153,Z 170.702,A -85,B 0,C 180,E1 -18325.886,E2 -18325.886} C_VEL
LIN {X 0,Y 263.128,Z 170.705,A -85,B 0,C 180,E1 -18329.504,E2 -18329.504} C_VEL
LIN {X 0,Y 263.144,Z 170.707,A -85,B 0,C 180,E1 -18332.997,E2 -18332.997} C_VEL
LIN {X 0,Y 263.146,Z 170.702,A -85,B 0,C 180,E1 -18336.383,E2 -18336.383} C_VEL
LIN {X 0,Y 263.211,Z 170.695,A -85,B 0,C 180,E1 -18339.689,E2 -18339.689} C_VEL
LIN {X 0,Y 263.291,Z 170.684,A -85,B 0,C 180,E1 -18344.518,E2 -18344.518} C_VEL
LIN {X 0,Y 263.351,Z 170.679,A -85,B 0,C 180,E1 -18349.233,E2 -18349.233} C_VEL
LIN {X 0,Y 263.529,Z 170.657,A -85,B 0,C 180,E1 -18352.337,E2 -18352.337} C_VEL
LIN {X 0,Y 263.737,Z 170.633,A -85,B 0,C 180,E1 -18358.473,E2 -18358.473} C_VEL
LIN {X 0,Y 263.71,Z 170.631,A -85,B 0,C 180,E1 -18360.843,E2 -18360.843} C_VEL
LIN {X 0,Y 263.027,Z 170.716,A -85,B 0,C 180,E1 -18362.114,E2 -18362.114} C_VEL
LIN {X 0,Y 260.06,Z 171.076,A -85,B 0,C 180,E1 -18364.182,E2 -18364.182} C_VEL
LIN {X 0,Y 257.558,Z 171.381,A -85,B 0,C 180,E1 -18365.864,E2 -18365.864} C_VEL
LIN {X 0,Y 256.521,Z 171.508,A -85,B 0,C 180,E1 -18367.172,E2 -18367.172} C_VEL
LIN {X 0,Y 256.456,Z 171.517,A -85,B 0,C 180,E1 -18367.616,E2 -18367.616} C_VEL
LIN {X 0,Y 256.273,Z 171.556,A -85,B 0,C 180,E1 -18371.068,E2 -18371.068} C_VEL
LIN {X 0,Y 256.215,Z 171.568,A -85,B 0,C 180,E1 -18375.92,E2 -18375.92} C_VEL
LIN {X 0,Y 256.12,Z 171.565,A -85,B 0,C 180,E1 -18381.097,E2 -18381.097} C_VEL
LIN {X 0,Y 256.084,Z 171.584,A -85,B 0,C 180,E1 -18385.087,E2 -18385.087} C_VEL
LIN {X 0,Y 256.078,Z 171.582,A -85,B 0,C 180,E1 -18388.569,E2 -18388.569} C_VEL
LIN {X 0,Y 256.072,Z 171.589,A -85,B 0,C 180,E1 -18391.699,E2 -18391.699} C_VEL
LIN {X 0,Y 256.081,Z 171.587,A -85,B 0,C 180,E1 -18395.193,E2 -18395.193} C_VEL
LIN {X 0,Y 256.112,Z 171.585,A -85,B 0,C 180,E1 -18397.269,E2 -18397.269} C_VEL
LIN {X 0,Y 256.02,Z 171.594,A -85,B 0,C 180,E1 -18401.21,E2 -18401.21} C_VEL
LIN {X 0,Y 256.019,Z 171.588,A -85,B 0,C 180,E1 -18405.539,E2 -18405.539} C_VEL
LIN {X 0,Y 256.019,Z 171.593,A -85,B 0,C 180,E1 -18408.789,E2 -18408.789} C_VEL
LIN {X 0,Y 256.127,Z 171.579,A -85,B 0,C 180,E1 -18412.866,E2 -18412.866} C_VEL
LIN {X 0,Y 256.152,Z 171.619,A -85,B 0,C 180,E1 -18414.577,E2 -18414.577} C_VEL
LIN {X 0,Y 258.245,Z 181.344,A -85,B 0,C 180,E1 -18418.295,E2 -18418.295} C_VEL
LIN {X 0,Y 259.347,Z 186.866,A -85,B 0,C 180,E1 -18420.322,E2 -18420.322} C_VEL
LIN {X 0,Y 265.052,Z 203.079,A -85,B 0,C 180,E1 -18421.426,E2 -18421.426} C_VEL
LIN {X 0,Y 269.451,Z 233.691,A -85,B 0,C 180,E1 -18422.79,E2 -18422.79} C_VEL
LIN {X 0,Y 267.407,Z 295.77,A -85,B 0,C 180,E1 -18424.561,E2 -18424.561} C_VEL
LIN {X 0,Y 266.429,Z 309.326,A -85,B 0,C 180,E1 -18425.244,E2 -18425.244} C_VEL
LIN {X 0,Y 265.112,Z 321.675,A -85,B 0,C 180,E1 -18426.154,E2 -18426.154} C_VEL
LIN {X 0,Y 263.41,Z 334.365,A -85,B 0,C 180,E1 -18427.447,E2 -18427.447} C_VEL
LIN {X 0,Y 261.65,Z 345.685,A -85,B 0,C 180,E1 -18428.945,E2 -18428.945} C_VEL
LIN {X 0,Y 260.007,Z 355.899,A -85,B 0,C 180,E1 -18430.663,E2 -18430.663} C_VEL
LIN {X 0,Y 258.489,Z 365.111,A -85,B 0,C 180,E1 -18432.598,E2 -18432.598} C_VEL
LIN {X 0,Y 256.918,Z 374.078,A -85,B 0,C 180,E1 -18434.937,E2 -18434.937} C_VEL
LIN {X 0,Y 255.592,Z 381.237,A -85,B 0,C 180,E1 -18437.292,E2 -18437.292} C_VEL
LIN {X 0,Y 254.801,Z 386.942,A -85,B 0,C 180,E1 -18439.672,E2 -18439.672} C_VEL
LIN {X 0,Y 254.306,Z 391.411,A -85,B 0,C 180,E1 -18442.057,E2 -18442.057} C_VEL
LIN {X 0,Y 254.022,Z 395.265,A -85,B 0,C 180,E1 -18444.881,E2 -18444.881} C_VEL
LIN {X 0,Y 253.993,Z 397.111,A -85,B 0,C 180,E1 -18446.828,E2 -18446.828} C_VEL
LIN {X 0,Y 254.025,Z 398.12,A -85,B 0,C 180,E1 -18448.415,E2 -18448.415} C_VEL
LIN {X 0,Y 254.054,Z 398.728,A -85,B 0,C 180,E1 -18450,E2 -18450} C_VEL
LIN {X 0,Y 254.014,Z 398.939,A -85,B 0,C 180,E1 -18451.585,E2 -18451.585} C_VEL
LIN {X 0,Y 253.949,Z 398.713,A -85,B 0,C 180,E1 -18453.173,E2 -18453.173} C_VEL
LIN {X 0,Y 253.99,Z 397.936,A -85,B 0,C 180,E1 -18455.039,E2 -18455.039} C_VEL
LIN {X 0,Y 254.318,Z 395.647,A -85,B 0,C 180,E1 -18457.942,E2 -18457.942} C_VEL
LIN {X 0,Y 254.94,Z 392.682,A -85,B 0,C 180,E1 -18460.323,E2 -18460.323} C_VEL
LIN {X 0,Y 255.867,Z 388.692,A -85,B 0,C 180,E1 -18462.694,E2 -18462.694} C_VEL
LIN {X 0,Y 257.28,Z 383.591,A -85,B 0,C 180,E1 -18465.041,E2 -18465.041} C_VEL
LIN {X 0,Y 259.119,Z 377.204,A -85,B 0,C 180,E1 -18467.359,E2 -18467.359} C_VEL
LIN {X 0,Y 261.065,Z 369.586,A -85,B 0,C 180,E1 -18469.572,E2 -18469.572} C_VEL
LIN {X 0,Y 263.251,Z 361.181,A -85,B 0,C 180,E1 -18471.536,E2 -18471.536} C_VEL
LIN {X 0,Y 265.752,Z 351.366,A -85,B 0,C 180,E1 -18473.371,E2 -18473.371} C_VEL
LIN {X 0,Y 268.169,Z 340.454,A -85,B 0,C 180,E1 -18474.999,E2 -18474.999} C_VEL
LIN {X 0,Y 270.653,Z 328.07,A -85,B 0,C 180,E1 -18476.403,E2 -18476.403} C_VEL
LIN {X 0,Y 272.533,Z 316.027,A -85,B 0,C 180,E1 -18477.449,E2 -18477.449} C_VEL
LIN {X 0,Y 274.194,Z 302.706,A -85,B 0,C 180,E1 -18478.254,E2 -18478.254} C_VEL
LIN {X 0,Y 275.201,Z 289.737,A -85,B 0,C 180,E1 -18478.766,E2 -18478.766} C_VEL
LIN {X 0,Y 277.461,Z 236.173,A -85,B 0,C 180,E1 -18480.27,E2 -18480.27} C_VEL
LIN {X 0,Y 274.598,Z 216.55,A -85,B 0,C 180,E1 -18481.388,E2 -18481.388} C_VEL
LIN {X 0,Y 273.363,Z 212.838,A -85,B 0,C 180,E1 -18481.713,E2 -18481.713} C_VEL
LIN {X 0,Y 266.695,Z 198.25,A -85,B 0,C 180,E1 -18483.362,E2 -18483.362} C_VEL
LIN {X 0,Y 261.637,Z 188.762,A -85,B 0,C 180,E1 -18484.651,E2 -18484.651} C_VEL
LIN {X 0,Y 259.805,Z 184.968,A -85,B 0,C 180,E1 -18485.214,E2 -18485.214} C_VEL
LIN {X 0,Y 258.268,Z 179.126,A -85,B 0,C 180,E1 -18487.894,E2 -18487.894} C_VEL
LIN {X 0,Y 256.036,Z 171.593,A -85,B 0,C 180,E1 -18491.722,E2 -18491.722} C_VEL
LIN {X 0,Y 256.019,Z 171.598,A -85,B 0,C 180,E1 -18495.54,E2 -18495.54} C_VEL
LIN {X 0,Y 256.041,Z 171.592,A -85,B 0,C 180,E1 -18498.794,E2 -18498.794} C_VEL
LIN {X 0,Y 256.127,Z 171.574,A -85,B 0,C 180,E1 -18502.867,E2 -18502.867} C_VEL
LIN {X 0,Y 256.067,Z 171.578,A -85,B 0,C 180,E1 -18506.707,E2 -18506.707} C_VEL
LIN {X 0,Y 256.042,Z 171.58,A -85,B 0,C 180,E1 -18510.391,E2 -18510.391} C_VEL
LIN {X 0,Y 256.06,Z 171.582,A -85,B 0,C 180,E1 -18513.951,E2 -18513.951} C_VEL
LIN {X 0,Y 256.059,Z 171.588,A -85,B 0,C 180,E1 -18517.402,E2 -18517.402} C_VEL
LIN {X 0,Y 256.105,Z 171.575,A -85,B 0,C 180,E1 -18520.774,E2 -18520.774} C_VEL
LIN {X 0,Y 256.216,Z 171.556,A -85,B 0,C 180,E1 -18524.08,E2 -18524.08} C_VEL
LIN {X 0,Y 256.273,Z 171.547,A -85,B 0,C 180,E1 -18528.932,E2 -18528.932} C_VEL
LIN {X 0,Y 256.502,Z 171.526,A -85,B 0,C 180,E1 -18532.126,E2 -18532.126} C_VEL
LIN {X 0,Y 256.447,Z 171.531,A -85,B 0,C 180,E1 -18536.858,E2 -18536.858} C_VEL
LIN {X 0,Y 256.697,Z 171.497,A -85,B 0,C 180,E1 -18538.431,E2 -18538.431} C_VEL
LIN {X 0,Y 256.697,Z 171.499,A -85,B 0,C 180,E1 -18541.569,E2 -18541.569} C_VEL
LIN {X 0,Y 256.449,Z 171.532,A -85,B 0,C 180,E1 -18546.576,E2 -18546.576} C_VEL
LIN {X 0,Y 256.405,Z 171.538,A -85,B 0,C 180,E1 -18549.466,E2 -18549.466} C_VEL
LIN {X 0,Y 256.209,Z 171.572,A -85,B 0,C 180,E1 -18554.293,E2 -18554.293} C_VEL
LIN {X 0,Y 256.149,Z 171.576,A -85,B 0,C 180,E1 -18557.566,E2 -18557.566} C_VEL
LIN {X 0,Y 256.172,Z 171.652,A -85,B 0,C 180,E1 -18560.475,E2 -18560.475} C_VEL
LIN {X 0,Y 257.293,Z 175.536,A -85,B 0,C 180,E1 -18562.41,E2 -18562.41} C_VEL
LIN {X 0,Y 259.9,Z 179.738,A -85,B 0,C 180,E1 -18563.105,E2 -18563.105} C_VEL
LIN {X 0,Y 267.098,Z 192.332,A -85,B 0,C 180,E1 -18564.937,E2 -18564.937} C_VEL
LIN {X 0,Y 273.922,Z 206.044,A -85,B 0,C 180,E1 -18566.586,E2 -18566.586} C_VEL
LIN {X 0,Y 278.341,Z 216.742,A -85,B 0,C 180,E1 -18567.643,E2 -18567.643} C_VEL
LIN {X 0,Y 275.22,Z 283.03,A -85,B 0,C 180,E1 -18569.508,E2 -18569.508} C_VEL
LIN {X 0,Y 274.007,Z 296.363,A -85,B 0,C 180,E1 -18570.169,E2 -18570.169} C_VEL
LIN {X 0,Y 272.65,Z 308.076,A -85,B 0,C 180,E1 -18571.033,E2 -18571.033} C_VEL
LIN {X 0,Y 270.813,Z 319.576,A -85,B 0,C 180,E1 -18572.149,E2 -18572.149} C_VEL
LIN {X 0,Y 268.559,Z 330.953,A -85,B 0,C 180,E1 -18573.577,E2 -18573.577} C_VEL
LIN {X 0,Y 266.381,Z 340.712,A -85,B 0,C 180,E1 -18575.126,E2 -18575.126} C_VEL
LIN {X 0,Y 264.024,Z 350.237,A -85,B 0,C 180,E1 -18577.006,E2 -18577.006} C_VEL
LIN {X 0,Y 261.924,Z 357.996,A -85,B 0,C 180,E1 -18578.909,E2 -18578.909} C_VEL
LIN {X 0,Y 259.725,Z 365.846,A -85,B 0,C 180,E1 -18581.331,E2 -18581.331} C_VEL
LIN {X 0,Y 257.875,Z 372.07,A -85,B 0,C 180,E1 -18583.772,E2 -18583.772} C_VEL
LIN {X 0,Y 256.533,Z 376.53,A -85,B 0,C 180,E1 -18586.016,E2 -18586.016} C_VEL
LIN {X 0,Y 255.365,Z 380.491,A -85,B 0,C 180,E1 -18588.661,E2 -18588.661} C_VEL
LIN {X 0,Y 254.695,Z 382.572,A -85,B 0,C 180,E1 -18590.605,E2 -18590.605} C_VEL
LIN {X 0,Y 254.025,Z 384.457,A -85,B 0,C 180,E1 -18593.354,E2 -18593.354} C_VEL
LIN {X 0,Y 253.685,Z 385.15,A -85,B 0,C 180,E1 -18596.353,E2 -18596.353} C_VEL
LIN {X 0,Y 253.631,Z 384.449,A -85,B 0,C 180,E1 -18599.204,E2 -18599.204} C_VEL
LIN {X 0,Y 253.96,Z 382.193,A -85,B 0,C 180,E1 -18602.321,E2 -18602.321} C_VEL
LIN {X 0,Y 254.428,Z 379.43,A -85,B 0,C 180,E1 -18604.649,E2 -18604.649} C_VEL
LIN {X 0,Y 255.057,Z 375.066,A -85,B 0,C 180,E1 -18607.309,E2 -18607.309} C_VEL
LIN {X 0,Y 255.982,Z 369.159,A -85,B 0,C 180,E1 -18609.985,E2 -18609.985} C_VEL
LIN {X 0,Y 257.252,Z 361.925,A -85,B 0,C 180,E1 -18612.511,E2 -18612.511} C_VEL
LIN {X 0,Y 258.649,Z 354.304,A -85,B 0,C 180,E1 -18614.637,E2 -18614.637} C_VEL
LIN {X 0,Y 260.114,Z 345.769,A -85,B 0,C 180,E1 -18616.578,E2 -18616.578} C_VEL
LIN {X 0,Y 261.77,Z 335.896,A -85,B 0,C 180,E1 -18618.383,E2 -18618.383} C_VEL
LIN {X 0,Y 263.431,Z 324.951,A -85,B 0,C 180,E1 -18619.982,E2 -18619.982} C_VEL
LIN {X 0,Y 264.863,Z 314.213,A -85,B 0,C 180,E1 -18621.224,E2 -18621.224} C_VEL
LIN {X 0,Y 266.104,Z 302.005,A -85,B 0,C 180,E1 -18622.316,E2 -18622.316} C_VEL
LIN {X 0,Y 267.232,Z 288.525,A -85,B 0,C 180,E1 -18623.156,E2 -18623.156} C_VEL
LIN {X 0,Y 267.94,Z 276.102,A -85,B 0,C 180,E1 -18623.647,E2 -18623.647} C_VEL
LIN {X 0,Y 270.111,Z 210.628,A -85,B 0,C 180,E1 -18625.469,E2 -18625.469} C_VEL
LIN {X 0,Y 268.905,Z 205.405,A -85,B 0,C 180,E1 -18625.742,E2 -18625.742} C_VEL
LIN {X 0,Y 262.377,Z 187.696,A -85,B 0,C 180,E1 -18626.929,E2 -18626.929} C_VEL
LIN {X 0,Y 257.108,Z 173.949,A -85,B 0,C 180,E1 -18627.944,E2 -18627.944} C_VEL
LIN {X 0,Y 256.679,Z 171.513,A -85,B 0,C 180,E1 -18628.921,E2 -18628.921} C_VEL
LIN {X 0,Y 256.703,Z 171.508,A -85,B 0,C 180,E1 -18631.569,E2 -18631.569} C_VEL
LIN {X 0,Y 256.457,Z 171.539,A -85,B 0,C 180,E1 -18636.293,E2 -18636.293} C_VEL
LIN {X 0,Y 256.429,Z 171.544,A -85,B 0,C 180,E1 -18639.465,E2 -18639.465} C_VEL
LIN {X 0,Y 256.214,Z 171.57,A -85,B 0,C 180,E1 -18644.293,E2 -18644.293} C_VEL
LIN {X 0,Y 256.171,Z 171.567,A -85,B 0,C 180,E1 -18647.565,E2 -18647.565} C_VEL
LIN {X 0,Y 256.14,Z 171.578,A -85,B 0,C 180,E1 -18651.108,E2 -18651.108} C_VEL
LIN {X 0,Y 256.087,Z 171.577,A -85,B 0,C 180,E1 -18655.089,E2 -18655.089} C_VEL
LIN {X 0,Y 256.092,Z 171.583,A -85,B 0,C 180,E1 -18658.575,E2 -18658.575} C_VEL
LIN {X 0,Y 256.076,Z 171.579,A -85,B 0,C 180,E1 -18661.701,E2 -18661.701} C_VEL
LIN {X 0,Y 256.082,Z 171.575,A -85,B 0,C 180,E1 -18665.193,E2 -18665.193} C_VEL
LIN {X 0,Y 256.112,Z 171.58,A -85,B 0,C 180,E1 -18667.269,E2 -18667.269} C_VEL
LIN {X 0,Y 256.042,Z 171.592,A -85,B 0,C 180,E1 -18671.206,E2 -18671.206} C_VEL
LIN {X 0,Y 256.019,Z 171.573,A -85,B 0,C 180,E1 -18675.54,E2 -18675.54} C_VEL
LIN {X 0,Y 256.02,Z 171.58,A -85,B 0,C 180,E1 -18678.789,E2 -18678.789} C_VEL
LIN {X 0,Y 256.13,Z 171.58,A -85,B 0,C 180,E1 -18682.867,E2 -18682.867} C_VEL
LIN {X 0,Y 256.068,Z 171.586,A -85,B 0,C 180,E1 -18686.707,E2 -18686.707} C_VEL
LIN {X 0,Y 256.057,Z 171.586,A -85,B 0,C 180,E1 -18690.393,E2 -18690.393} C_VEL
LIN {X 0,Y 256.135,Z 171.577,A -85,B 0,C 180,E1 -18694.888,E2 -18694.888} C_VEL
LIN {X 0,Y 256.126,Z 171.579,A -85,B 0,C 180,E1 -18699.101,E2 -18699.101} C_VEL
LIN {X 0,Y 256.215,Z 171.566,A -85,B 0,C 180,E1 -18704.08,E2 -18704.08} C_VEL
LIN {X 0,Y 256.29,Z 171.559,A -85,B 0,C 180,E1 -18708.933,E2 -18708.933} C_VEL
LIN {X 0,Y 256.493,Z 171.535,A -85,B 0,C 180,E1 -18712.126,E2 -18712.126} C_VEL
LIN {X 0,Y 256.454,Z 171.538,A -85,B 0,C 180,E1 -18716.858,E2 -18716.858} C_VEL
LIN {X 0,Y 256.699,Z 171.51,A -85,B 0,C 180,E1 -18718.431,E2 -18718.431} C_VEL
LIN {X 0,Y 256.699,Z 171.506,A -85,B 0,C 180,E1 -18721.569,E2 -18721.569} C_VEL
LIN {X 0,Y 256.456,Z 171.517,A -85,B 0,C 180,E1 -18727.616,E2 -18727.616} C_VEL
LIN {X 0,Y 255.802,Z 171.609,A -85,B 0,C 180,E1 -18728.925,E2 -18728.925} C_VEL
LIN {X 0,Y 252.815,Z 171.987,A -85,B 0,C 180,E1 -18731.052,E2 -18731.052} C_VEL
LIN {X 0,Y 250.27,Z 172.308,A -85,B 0,C 180,E1 -18732.785,E2 -18732.785} C_VEL
LIN {X 0,Y 249.207,Z 172.443,A -85,B 0,C 180,E1 -18734.134,E2 -18734.134} C_VEL
LIN {X 0,Y 249.139,Z 172.448,A -85,B 0,C 180,E1 -18734.591,E2 -18734.591} C_VEL
LIN {X 0,Y 249.078,Z 172.448,A -85,B 0,C 180,E1 -18738.082,E2 -18738.082} C_VEL
LIN {X 0,Y 249.044,Z 172.448,A -85,B 0,C 180,E1 -18741.522,E2 -18741.522} C_VEL
LIN {X 0,Y 249.045,Z 172.463,A -85,B 0,C 180,E1 -18745.439,E2 -18745.439} C_VEL
LIN {X 0,Y 249.025,Z 172.461,A -85,B 0,C 180,E1 -18748.968,E2 -18748.968} C_VEL
LIN {X 0,Y 249.027,Z 172.464,A -85,B 0,C 180,E1 -18752.426,E2 -18752.426} C_VEL
LIN {X 0,Y 249.028,Z 172.465,A -85,B 0,C 180,E1 -18756.346,E2 -18756.346} C_VEL
LIN {X 0,Y 248.98,Z 172.47,A -85,B 0,C 180,E1 -18760.483,E2 -18760.483} C_VEL
LIN {X 0,Y 248.963,Z 172.469,A -85,B 0,C 180,E1 -18764.888,E2 -18764.888} C_VEL
LIN {X 0,Y 248.98,Z 172.472,A -85,B 0,C 180,E1 -18767.355,E2 -18767.355} C_VEL
LIN {X 0,Y 249.041,Z 172.463,A -85,B 0,C 180,E1 -18772.201,E2 -18772.201} C_VEL
LIN {X 0,Y 249.109,Z 172.614,A -85,B 0,C 180,E1 -18774.079,E2 -18774.079} C_VEL
LIN {X 0,Y 251.191,Z 182.272,A -85,B 0,C 180,E1 -18777.886,E2 -18777.886} C_VEL
LIN {X 0,Y 252.157,Z 186.763,A -85,B 0,C 180,E1 -18779.583,E2 -18779.583} C_VEL
LIN {X 0,Y 258.728,Z 204.976,A -85,B 0,C 180,E1 -18780.866,E2 -18780.866} C_VEL
LIN {X 0,Y 262.902,Z 234.516,A -85,B 0,C 180,E1 -18782.221,E2 -18782.221} C_VEL
LIN {X 0,Y 260.772,Z 296.064,A -85,B 0,C 180,E1 -18784.027,E2 -18784.027} C_VEL
LIN {X 0,Y 259.742,Z 309.45,A -85,B 0,C 180,E1 -18784.722,E2 -18784.722} C_VEL
LIN {X 0,Y 258.326,Z 322.208,A -85,B 0,C 180,E1 -18785.701,E2 -18785.701} C_VEL
LIN {X 0,Y 256.588,Z 334.738,A -85,B 0,C 180,E1 -18787.026,E2 -18787.026} C_VEL
LIN {X 0,Y 254.78,Z 345.956,A -85,B 0,C 180,E1 -18788.562,E2 -18788.562} C_VEL
LIN {X 0,Y 253.267,Z 355.058,A -85,B 0,C 180,E1 -18790.127,E2 -18790.127} C_VEL
LIN {X 0,Y 251.656,Z 364.389,A -85,B 0,C 180,E1 -18792.109,E2 -18792.109} C_VEL
LIN {X 0,Y 250.023,Z 373.447,A -85,B 0,C 180,E1 -18794.512,E2 -18794.512} C_VEL
LIN {X 0,Y 248.633,Z 380.71,A -85,B 0,C 180,E1 -18796.93,E2 -18796.93} C_VEL
LIN {X 0,Y 247.787,Z 386.49,A -85,B 0,C 180,E1 -18799.376,E2 -18799.376} C_VEL
LIN {X 0,Y 247.256,Z 391.02,A -85,B 0,C 180,E1 -18801.829,E2 -18801.829} C_VEL
LIN {X 0,Y 246.944,Z 395.153,A -85,B 0,C 180,E1 -18804.937,E2 -18804.937} C_VEL
LIN {X 0,Y 246.893,Z 396.827,A -85,B 0,C 180,E1 -18806.736,E2 -18806.736} C_VEL
LIN {X 0,Y 246.934,Z 397.862,A -85,B 0,C 180,E1 -18808.369,E2 -18808.369} C_VEL
LIN {X 0,Y 246.983,Z 398.496,A -85,B 0,C 180,E1 -18810,E2 -18810} C_VEL
LIN {X 0,Y 246.921,Z 398.731,A -85,B 0,C 180,E1 -18811.631,E2 -18811.631} C_VEL
LIN {X 0,Y 246.853,Z 398.553,A -85,B 0,C 180,E1 -18813.264,E2 -18813.264} C_VEL
LIN {X 0,Y 247.01,Z 396.952,A -85,B 0,C 180,E1 -18816.535,E2 -18816.535} C_VEL
LIN {X 0,Y 247.272,Z 395.565,A -85,B 0,C 180,E1 -18818.17,E2 -18818.17} C_VEL
LIN {X 0,Y 247.918,Z 392.66,A -85,B 0,C 180,E1 -18820.618,E2 -18820.618} C_VEL
LIN {X 0,Y 248.909,Z 388.738,A -85,B 0,C 180,E1 -18823.055,E2 -18823.055} C_VEL
LIN {X 0,Y 250.427,Z 383.699,A -85,B 0,C 180,E1 -18825.463,E2 -18825.463} C_VEL
LIN {X 0,Y 252.34,Z 377.396,A -85,B 0,C 180,E1 -18827.84,E2 -18827.84} C_VEL
LIN {X 0,Y 254.521,Z 369.409,A -85,B 0,C 180,E1 -18830.232,E2 -18830.232} C_VEL
LIN {X 0,Y 257.152,Z 359.792,A -85,B 0,C 180,E1 -18832.496,E2 -18832.496} C_VEL
LIN {X 0,Y 259.847,Z 349.73,A -85,B 0,C 180,E1 -18834.36,E2 -18834.36} C_VEL
LIN {X 0,Y 262.45,Z 338.42,A -85,B 0,C 180,E1 -18836.008,E2 -18836.008} C_VEL
LIN {X 0,Y 264.666,Z 327.401,A -85,B 0,C 180,E1 -18837.262,E2 -18837.262} C_VEL
LIN {X 0,Y 266.676,Z 315.239,A -85,B 0,C 180,E1 -18838.319,E2 -18838.319} C_VEL
LIN {X 0,Y 268.318,Z 302.544,A -85,B 0,C 180,E1 -18839.092,E2 -18839.092} C_VEL
LIN {X 0,Y 269.34,Z 289.63,A -85,B 0,C 180,E1 -18839.614,E2 -18839.614} C_VEL
LIN {X 0,Y 271.651,Z 236.974,A -85,B 0,C 180,E1 -18841.123,E2 -18841.123} C_VEL
LIN {X 0,Y 268.96,Z 218.37,A -85,B 0,C 180,E1 -18842.224,E2 -18842.224} C_VEL
LIN {X 0,Y 262.933,Z 204.44,A -85,B 0,C 180,E1 -18843.802,E2 -18843.802} C_VEL
LIN {X 0,Y 257.328,Z 193.588,A -85,B 0,C 180,E1 -18845.296,E2 -18845.296} C_VEL
LIN {X 0,Y 254.506,Z 188.601,A -85,B 0,C 180,E1 -18846.079,E2 -18846.079} C_VEL
LIN {X 0,Y 252.5,Z 184.711,A -85,B 0,C 180,E1 -18846.714,E2 -18846.714} C_VEL
LIN {X 0,Y 250.54,Z 177.754,A -85,B 0,C 180,E1 -18850.18,E2 -18850.18} C_VEL
LIN {X 0,Y 248.995,Z 172.475,A -85,B 0,C 180,E1 -18853.06,E2 -18853.06} C_VEL
LIN {X 0,Y 248.994,Z 172.465,A -85,B 0,C 180,E1 -18857.358,E2 -18857.358} C_VEL
LIN {X 0,Y 249.042,Z 172.461,A -85,B 0,C 180,E1 -18862.202,E2 -18862.202} C_VEL
LIN {X 0,Y 249.045,Z 172.461,A -85,B 0,C 180,E1 -18865.64,E2 -18865.64} C_VEL
LIN {X 0,Y 248.996,Z 172.466,A -85,B 0,C 180,E1 -18869.465,E2 -18869.465} C_VEL
LIN {X 0,Y 249.012,Z 172.465,A -85,B 0,C 180,E1 -18873.155,E2 -18873.155} C_VEL
LIN {X 0,Y 249.007,Z 172.464,A -85,B 0,C 180,E1 -18876.725,E2 -18876.725} C_VEL
LIN {X 0,Y 249.042,Z 172.45,A -85,B 0,C 180,E1 -18880.206,E2 -18880.206} C_VEL
LIN {X 0,Y 249.16,Z 172.437,A -85,B 0,C 180,E1 -18883.616,E2 -18883.616} C_VEL
LIN {X 0,Y 249.218,Z 172.426,A -85,B 0,C 180,E1 -18888.615,E2 -18888.615} C_VEL
LIN {X 0,Y 249.441,Z 172.408,A -85,B 0,C 180,E1 -18891.902,E2 -18891.902} C_VEL
LIN {X 0,Y 249.261,Z 172.432,A -85,B 0,C 180,E1 -18895.148,E2 -18895.148} C_VEL
LIN {X 0,Y 249.658,Z 172.373,A -85,B 0,C 180,E1 -18898.387,E2 -18898.387} C_VEL
LIN {X 0,Y 249.658,Z 172.375,A -85,B 0,C 180,E1 -18901.613,E2 -18901.613} C_VEL
LIN {X 0,Y 249.426,Z 172.407,A -85,B 0,C 180,E1 -18906.557,E2 -18906.557} C_VEL
LIN {X 0,Y 249.335,Z 172.419,A -85,B 0,C 180,E1 -18909.737,E2 -18909.737} C_VEL
LIN {X 0,Y 249.152,Z 172.449,A -85,B 0,C 180,E1 -18914.707,E2 -18914.707} C_VEL
LIN {X 0,Y 249.081,Z 172.455,A -85,B 0,C 180,E1 -18918.082,E2 -18918.082} C_VEL
LIN {X 0,Y 249.09,Z 172.608,A -85,B 0,C 180,E1 -18919.147,E2 -18919.147} C_VEL
LIN {X 0,Y 250.006,Z 175.729,A -85,B 0,C 180,E1 -18920.842,E2 -18920.842} C_VEL
LIN {X 0,Y 252.711,Z 180.049,A -85,B 0,C 180,E1 -18921.63,E2 -18921.63} C_VEL
LIN {X 0,Y 258.702,Z 189.923,A -85,B 0,C 180,E1 -18923.281,E2 -18923.281} C_VEL
LIN {X 0,Y 265.427,Z 202.549,A -85,B 0,C 180,E1 -18925.026,E2 -18925.026} C_VEL
LIN {X 0,Y 270.796,Z 214.385,A -85,B 0,C 180,E1 -18926.385,E2 -18926.385} C_VEL
LIN {X 0,Y 272.56,Z 219.027,A -85,B 0,C 180,E1 -18926.833,E2 -18926.833} C_VEL
LIN {X 0,Y 269.361,Z 283.448,A -85,B 0,C 180,E1 -18928.678,E2 -18928.678} C_VEL
LIN {X 0,Y 268.09,Z 296.714,A -85,B 0,C 180,E1 -18929.348,E2 -18929.348} C_VEL
LIN {X 0,Y 266.559,Z 309.129,A -85,B 0,C 180,E1 -18930.29,E2 -18930.29} C_VEL
LIN {X 0,Y 264.624,Z 320.498,A -85,B 0,C 180,E1 -18931.439,E2 -18931.439} C_VEL
LIN {X 0,Y 262.31,Z 331.589,A -85,B 0,C 180,E1 -18932.876,E2 -18932.876} C_VEL
LIN {X 0,Y 259.803,Z 342.16,A -85,B 0,C 180,E1 -18934.616,E2 -18934.616} C_VEL
LIN {X 0,Y 257.144,Z 352.167,A -85,B 0,C 180,E1 -18936.726,E2 -18936.726} C_VEL
LIN {X 0,Y 254.856,Z 360.144,A -85,B 0,C 180,E1 -18938.827,E2 -18938.827} C_VEL
LIN {X 0,Y 252.604,Z 367.626,A -85,B 0,C 180,E1 -18941.305,E2 -18941.305} C_VEL
LIN {X 0,Y 250.616,Z 373.89,A -85,B 0,C 180,E1 -18944.013,E2 -18944.013} C_VEL
LIN {X 0,Y 249.3,Z 377.998,A -85,B 0,C 180,E1 -18946.317,E2 -18946.317} C_VEL
LIN {X 0,Y 248.028,Z 381.887,A -85,B 0,C 180,E1 -18949.328,E2 -18949.328} C_VEL
LIN {X 0,Y 247.402,Z 383.632,A -85,B 0,C 180,E1 -18951.32,E2 -18951.32} C_VEL
LIN {X 0,Y 246.955,Z 384.756,A -85,B 0,C 180,E1 -18953.299,E2 -18953.299} C_VEL
LIN {X 0,Y 246.637,Z 385.317,A -85,B 0,C 180,E1 -18955.728,E2 -18955.728} C_VEL
LIN {X 0,Y 246.524,Z 384.801,A -85,B 0,C 180,E1 -18958.788,E2 -18958.788} C_VEL
LIN {X 0,Y 246.797,Z 382.698,A -85,B 0,C 180,E1 -18961.98,E2 -18961.98} C_VEL
LIN {X 0,Y 247.347,Z 379.546,A -85,B 0,C 180,E1 -18964.773,E2 -18964.773} C_VEL
LIN {X 0,Y 248.018,Z 375.151,A -85,B 0,C 180,E1 -18967.508,E2 -18967.508} C_VEL
LIN {X 0,Y 248.968,Z 369.346,A -85,B 0,C 180,E1 -18970.2,E2 -18970.2} C_VEL
LIN {X 0,Y 250.238,Z 362.321,A -85,B 0,C 180,E1 -18972.727,E2 -18972.727} C_VEL
LIN {X 0,Y 251.769,Z 354.265,A -85,B 0,C 180,E1 -18975.036,E2 -18975.036} C_VEL
LIN {X 0,Y 253.42,Z 344.908,A -85,B 0,C 180,E1 -18977.181,E2 -18977.181} C_VEL
LIN {X 0,Y 255.253,Z 334.425,A -85,B 0,C 180,E1 -18979.089,E2 -18979.089} C_VEL
LIN {X 0,Y 257.017,Z 322.869,A -85,B 0,C 180,E1 -18980.755,E2 -18980.755} C_VEL
LIN {X 0,Y 258.559,Z 310.793,A -85,B 0,C 180,E1 -18982.091,E2 -18982.091} C_VEL
LIN {X 0,Y 259.791,Z 298.629,A -85,B 0,C 180,E1 -18983.105,E2 -18983.105} C_VEL
LIN {X 0,Y 260.821,Z 285.809,A -85,B 0,C 180,E1 -18983.849,E2 -18983.849} C_VEL
LIN {X 0,Y 261.556,Z 269.27,A -85,B 0,C 180,E1 -18984.412,E2 -18984.412} C_VEL
LIN {X 0,Y 263.536,Z 211.269,A -85,B 0,C 180,E1 -18986.064,E2 -18986.064} C_VEL
LIN {X 0,Y 261.47,Z 204.309,A -85,B 0,C 180,E1 -18986.487,E2 -18986.487} C_VEL
LIN {X 0,Y 254.444,Z 185.806,A -85,B 0,C 180,E1 -18987.809,E2 -18987.809} C_VEL
LIN {X 0,Y 250.024,Z 174.189,A -85,B 0,C 180,E1 -18988.691,E2 -18988.691} C_VEL
LIN {X 0,Y 249.633,Z 172.392,A -85,B 0,C 180,E1 -18989.496,E2 -18989.496} C_VEL
LIN {X 0,Y 249.663,Z 172.385,A -85,B 0,C 180,E1 -18991.613,E2 -18991.613} C_VEL
LIN {X 0,Y 249.431,Z 172.413,A -85,B 0,C 180,E1 -18996.471,E2 -18996.471} C_VEL
LIN {X 0,Y 249.344,Z 172.428,A -85,B 0,C 180,E1 -18999.736,E2 -18999.736} C_VEL
LIN {X 0,Y 249.158,Z 172.447,A -85,B 0,C 180,E1 -19004.706,E2 -19004.706} C_VEL
LIN {X 0,Y 249.107,Z 172.452,A -85,B 0,C 180,E1 -19008.08,E2 -19008.08} C_VEL
LIN {X 0,Y 249.079,Z 172.459,A -85,B 0,C 180,E1 -19011.519,E2 -19011.519} C_VEL
LIN {X 0,Y 249.049,Z 172.454,A -85,B 0,C 180,E1 -19015.442,E2 -19015.442} C_VEL
LIN {X 0,Y 249.038,Z 172.462,A -85,B 0,C 180,E1 -19018.974,E2 -19018.974} C_VEL
LIN {X 0,Y 249.029,Z 172.452,A -85,B 0,C 180,E1 -19022.426,E2 -19022.426} C_VEL
LIN {X 0,Y 249.047,Z 172.457,A -85,B 0,C 180,E1 -19026.343,E2 -19026.343} C_VEL
LIN {X 0,Y 248.986,Z 172.468,A -85,B 0,C 180,E1 -19030.482,E2 -19030.482} C_VEL
LIN {X 0,Y 248.964,Z 172.456,A -85,B 0,C 180,E1 -19034.889,E2 -19034.889} C_VEL
LIN {X 0,Y 248.981,Z 172.449,A -85,B 0,C 180,E1 -19037.355,E2 -19037.355} C_VEL
LIN {X 0,Y 249.043,Z 172.46,A -85,B 0,C 180,E1 -19042.201,E2 -19042.201} C_VEL
LIN {X 0,Y 249.045,Z 172.46,A -85,B 0,C 180,E1 -19045.639,E2 -19045.639} C_VEL
LIN {X 0,Y 249.004,Z 172.465,A -85,B 0,C 180,E1 -19049.466,E2 -19049.466} C_VEL
LIN {X 0,Y 249.038,Z 172.463,A -85,B 0,C 180,E1 -19053.158,E2 -19053.158} C_VEL
LIN {X 0,Y 249.054,Z 172.456,A -85,B 0,C 180,E1 -19056.73,E2 -19056.73} C_VEL
LIN {X 0,Y 249.047,Z 172.461,A -85,B 0,C 180,E1 -19060.206,E2 -19060.206} C_VEL
LIN {X 0,Y 249.16,Z 172.444,A -85,B 0,C 180,E1 -19063.616,E2 -19063.616} C_VEL
LIN {X 0,Y 249.232,Z 172.441,A -85,B 0,C 180,E1 -19068.615,E2 -19068.615} C_VEL
LIN {X 0,Y 249.438,Z 172.412,A -85,B 0,C 180,E1 -19071.901,E2 -19071.901} C_VEL
LIN {X 0,Y 249.265,Z 172.429,A -85,B 0,C 180,E1 -19075.148,E2 -19075.148} C_VEL
LIN {X 0,Y 249.66,Z 172.387,A -85,B 0,C 180,E1 -19078.387,E2 -19078.387} C_VEL
LIN {X 0,Y 249.66,Z 172.382,A -85,B 0,C 180,E1 -19081.613,E2 -19081.613} C_VEL
LIN {X 0,Y 249.4,Z 172.394,A -85,B 0,C 180,E1 -19087.623,E2 -19087.623} C_VEL
LIN {X 0,Y 249.334,Z 172.415,A -85,B 0,C 180,E1 -19089.737,E2 -19089.737} C_VEL
LIN {X 0,Y 249.139,Z 172.448,A -85,B 0,C 180,E1 -19094.591,E2 -19094.591} C_VEL
LIN {X 0,Y 248.513,Z 172.53,A -85,B 0,C 180,E1 -19095.939,E2 -19095.939} C_VEL
